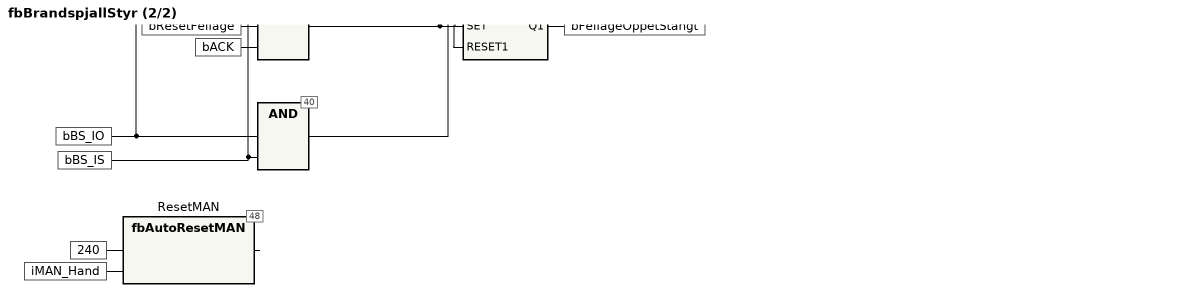
_CFC_ (* Continuous Function Chart, elements in execution order *)
(* **********************************************MOTIONERING********************************************** *)
(* **********************************************FELLÄGE SPJÄLL********************************************** *)
#0 OR(bManover, MotionManover)
#1 DELAY1:fbDelayedAlarmMinutes(_bLarm: bKomfel, _iMinutes: iKomfel_FL)
#2 AND(#0, NOT #1.bDelayedAlarm, NOT BrytManover)
#3 OVERRIDE:fbManualOverride(_bAuto: #2, _iMAN: iMAN_Hand, _iLM_Delay: iMAN_FL)
#4 bLM <= #3._bLM_DELAYED
#5 AND(#3._bStart, NOT bBRAND)
#6 bManoverUt <= #5
#7 PulsaMotionsKommando:TP(IN: bMotion, PT: t#1s)
#8 bResetFellage <= #7.Q
#9 AND(bManover, NOT bBRAND, #7.Q)
#10 DelayResetMotion:TON(IN: NOT bMotion, PT: t#15m)
#11 OR(bBRAND, #10.Q, bAvslutaMot)
#12 Motion_oppet:RS(SET: #9, RESET1: #11)
#13 StartaMotionOppetSpjall <= #12.Q1
#14 AND(NOT bManover, NOT bBRAND, #7.Q)
#15 OR(bBRAND, #10.Q, bAvslutaMot)
#16 Motion_stangt:RS(SET: #14, RESET1: #15)
#17 StartaMotionStangtSpjall <= #16.Q1
#18 OR(#12.Q1, #16.Q1)
#19 bMotionAktiv <= #18
#20 DelayMotOppet:TON(IN: StartaMotionOppetSpjall, PT: t#1s)
#21 Trig_bryt_man:R_TRIG(CLK: #20.Q)
#22 OR(bFellageStangerEJ, bBS_IS)
#23 DelayResetMotOppet:TON(IN: #22, PT: t#1s)
#24 Motion_oppet_bryt:SR(SET1: #21.Q, RESET: #23.Q)
#25 BrytManover <= #24.Q1
#26 AND(#24.Q1, #22)
#27 DelayMotStangt:TON(IN: StartaMotionStangtSpjall, PT: t#1s)
#28 Trig_man:R_TRIG(CLK: #27.Q)
#29 OR(bFellageOppnarEJ, bBS_IO)
#30 DelayResetMotStangt:TON(IN: #29, PT: t#1s)
#31 Motion_stangt_manover:SR(SET1: #28.Q, RESET: #30.Q)
#32 MotionManover <= #31.Q1
#33 AND(#31.Q1, #29)
#34 OR(#26, #33)
#35 bAvslutaMot <= #34
#36 AND(bManoverUt, NOT bBS_IO)
#37 DELAY2:fbDelayedAlarmSeconds(_bLarm: #36, _iSeconds: iBS_IO_FL)
#38 AND(NOT bManoverUt, NOT bBS_IS)
#39 DELAY3:fbDelayedAlarmSeconds(_bLarm: #38, _iSeconds: iBS_IS_FL)
#40 AND(bBS_IO, bBS_IS)
#41 OR(bResetFellage, bACK)
#42 SETRES1:RS(SET: #37.fDelayedAlarm2, RESET1: #41)
#43 bFellageOppnarEJ <= #42.Q1
#44 SETRES2:RS(SET: #39.fDelayedAlarm2, RESET1: #41)
#45 bFellageStangerEJ <= #44.Q1
#46 SETRES3:RS(SET: #40, RESET1: #41)
#47 bFellageOppetStangt <= #46.Q1
#48 ResetMAN:fbAutoResetMAN(240, iMAN_Hand)
_END_CFC_
END_FUNCTION_BLOCK

(* POU xEgna Funktionsblock/fbAutoResetMAN, CFC *)
FUNCTION_BLOCK fbAutoResetMAN
VAR_IN_OUT
	iMAN				:INT;

END_VAR
VAR_INPUT
	iResetDelay		:INT;

END_VAR
VAR_OUTPUT
END_VAR
VAR
	ResetDelay: TON;
END_VAR
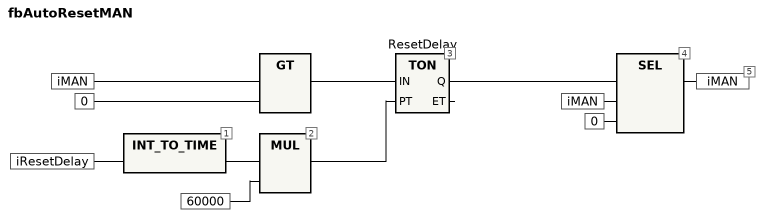
_CFC_ (* Continuous Function Chart, elements in execution order *)
#0 GT(iMAN, 0)
#1 INT_TO_TIME(iResetDelay)
#2 MUL(#1, 60000)
#3 ResetDelay:TON(IN: #0, PT: #2)
#4 SEL(#3.Q, iMAN, 0)
#5 iMAN <= #4
_END_CFC_
(* the same logic as Structured Text *)
ResetDelay(IN := iMAN > 0, PT := INT_TO_TIME(iResetDelay) * 60000);
iMAN := SEL(ResetDelay.Q, iMAN, 0);
END_FUNCTION_BLOCK

(* POU SYSTEM/Brandspjäll/HD71_BS201_BS202/HUS2_AS01_LB03_BS201_202, FAI *)
PROGRAM HUS2_AS01_LB03_BS201_202

VAR_INPUT
	bManover	 	:BOOL;
	bBRAND		:BOOL;
	bMotion		:BOOL;
	bKomfel		:BOOL;
END_VAR

VAR
	_bSetDefaultLocal: BOOL;

	SetAlarmDelay: FB_HVACPersistent_Int;
	SetAlarmDelay2: FB_HVACPersistent_Int;
	SetAlarmDelay3: FB_HVACPersistent_Int;
	SetAlarmDelay4: FB_HVACPersistent_Int;

	SpjallStyr: fbBrandspjallStyr2BS;

	ResetACK: fbBool_Reset;
	ResetACK2: fbBool_Reset;


END_VAR
(* body not read: cfc116 *)
END_PROGRAM

(* POU xEgna Funktionsblock/fbBrandspjallStyr2BS, CFC *)
FUNCTION_BLOCK fbBrandspjallStyr2BS
VAR_INPUT
	bManover						:BOOL;

	iMAN_FL1					:INT;
	bBS_IO1						:BOOL;
	iBS_IO_FL1					:INT;
	bBS_IS1						:BOOL;
	iBS_IS_FL1					:INT;
	bACK1						:BOOL;

	iMAN_FL2					:INT;
	bBS_IO2						:BOOL;
	iBS_IO_FL2					:INT;
	bBS_IS2						:BOOL;
	iBS_IS_FL2					:INT;
	bACK2						:BOOL;

	bBRAND						:BOOL;
	bKomfel						:BOOL;
	iKomfel_FL					:INT;
	bMotion						:BOOL;


END_VAR

VAR_IN_OUT
	iMAN_Hand1					:INT;
	iMAN_Hand2					:INT;
END_VAR

VAR_OUTPUT
	bManoverUt					:BOOL;
	bMotionAktiv					:BOOL;
	bLM1							:BOOL;
	bFellageOppnarEJ1			:BOOL;
	bFellageStangerEJ1			:BOOL;
	bFellageOppetStangt1			:BOOL;
	bLM2							:BOOL;
	bFellageOppnarEJ2			:BOOL;
	bFellageStangerEJ2			:BOOL;
	bFellageOppetStangt2			:BOOL;

END_VAR

VAR

	BrytManover: BOOL;
	MotionManover: BOOL;
	StartaMotionOppetSpjall: BOOL;
	StartaMotionStangtSpjall: BOOL;
	bResetFellage: BOOL;
	bAvslutaMot: BOOL;

	OVERRIDE1: fbManualOverride;
	ResetMAN1: fbAutoResetMAN;
	OVERRIDE2: fbManualOverride;
	ResetMAN2: fbAutoResetMAN;
	PulsaMotionsKommando: TP;
	DelayResetMotion: TON;

	DELAY1: fbDelayedAlarmMinutes;
	DELAY2: fbDelayedAlarmSeconds;
	DELAY3: fbDelayedAlarmSeconds;
	DELAY4: fbDelayedAlarmSeconds;
	DELAY5: fbDelayedAlarmSeconds;

	SETRES1: RS;
	SETRES2: RS;
	SETRES3: RS;
	SETRES4: RS;
	SETRES5: RS;
	SETRES6: RS;

	Motion_oppet: RS;
	Motion_oppet_bryt: SR;
	DelayMotOppet: TON;
	Trig_bryt_man: R_TRIG;
	DelayResetMotOppet: TON;

	Motion_stangt: RS;
	Motion_stangt_manover: SR;
	DelayMotStangt: TON;
	Trig_man: R_TRIG;
	DelayResetMotStangt: TON;


END_VAR
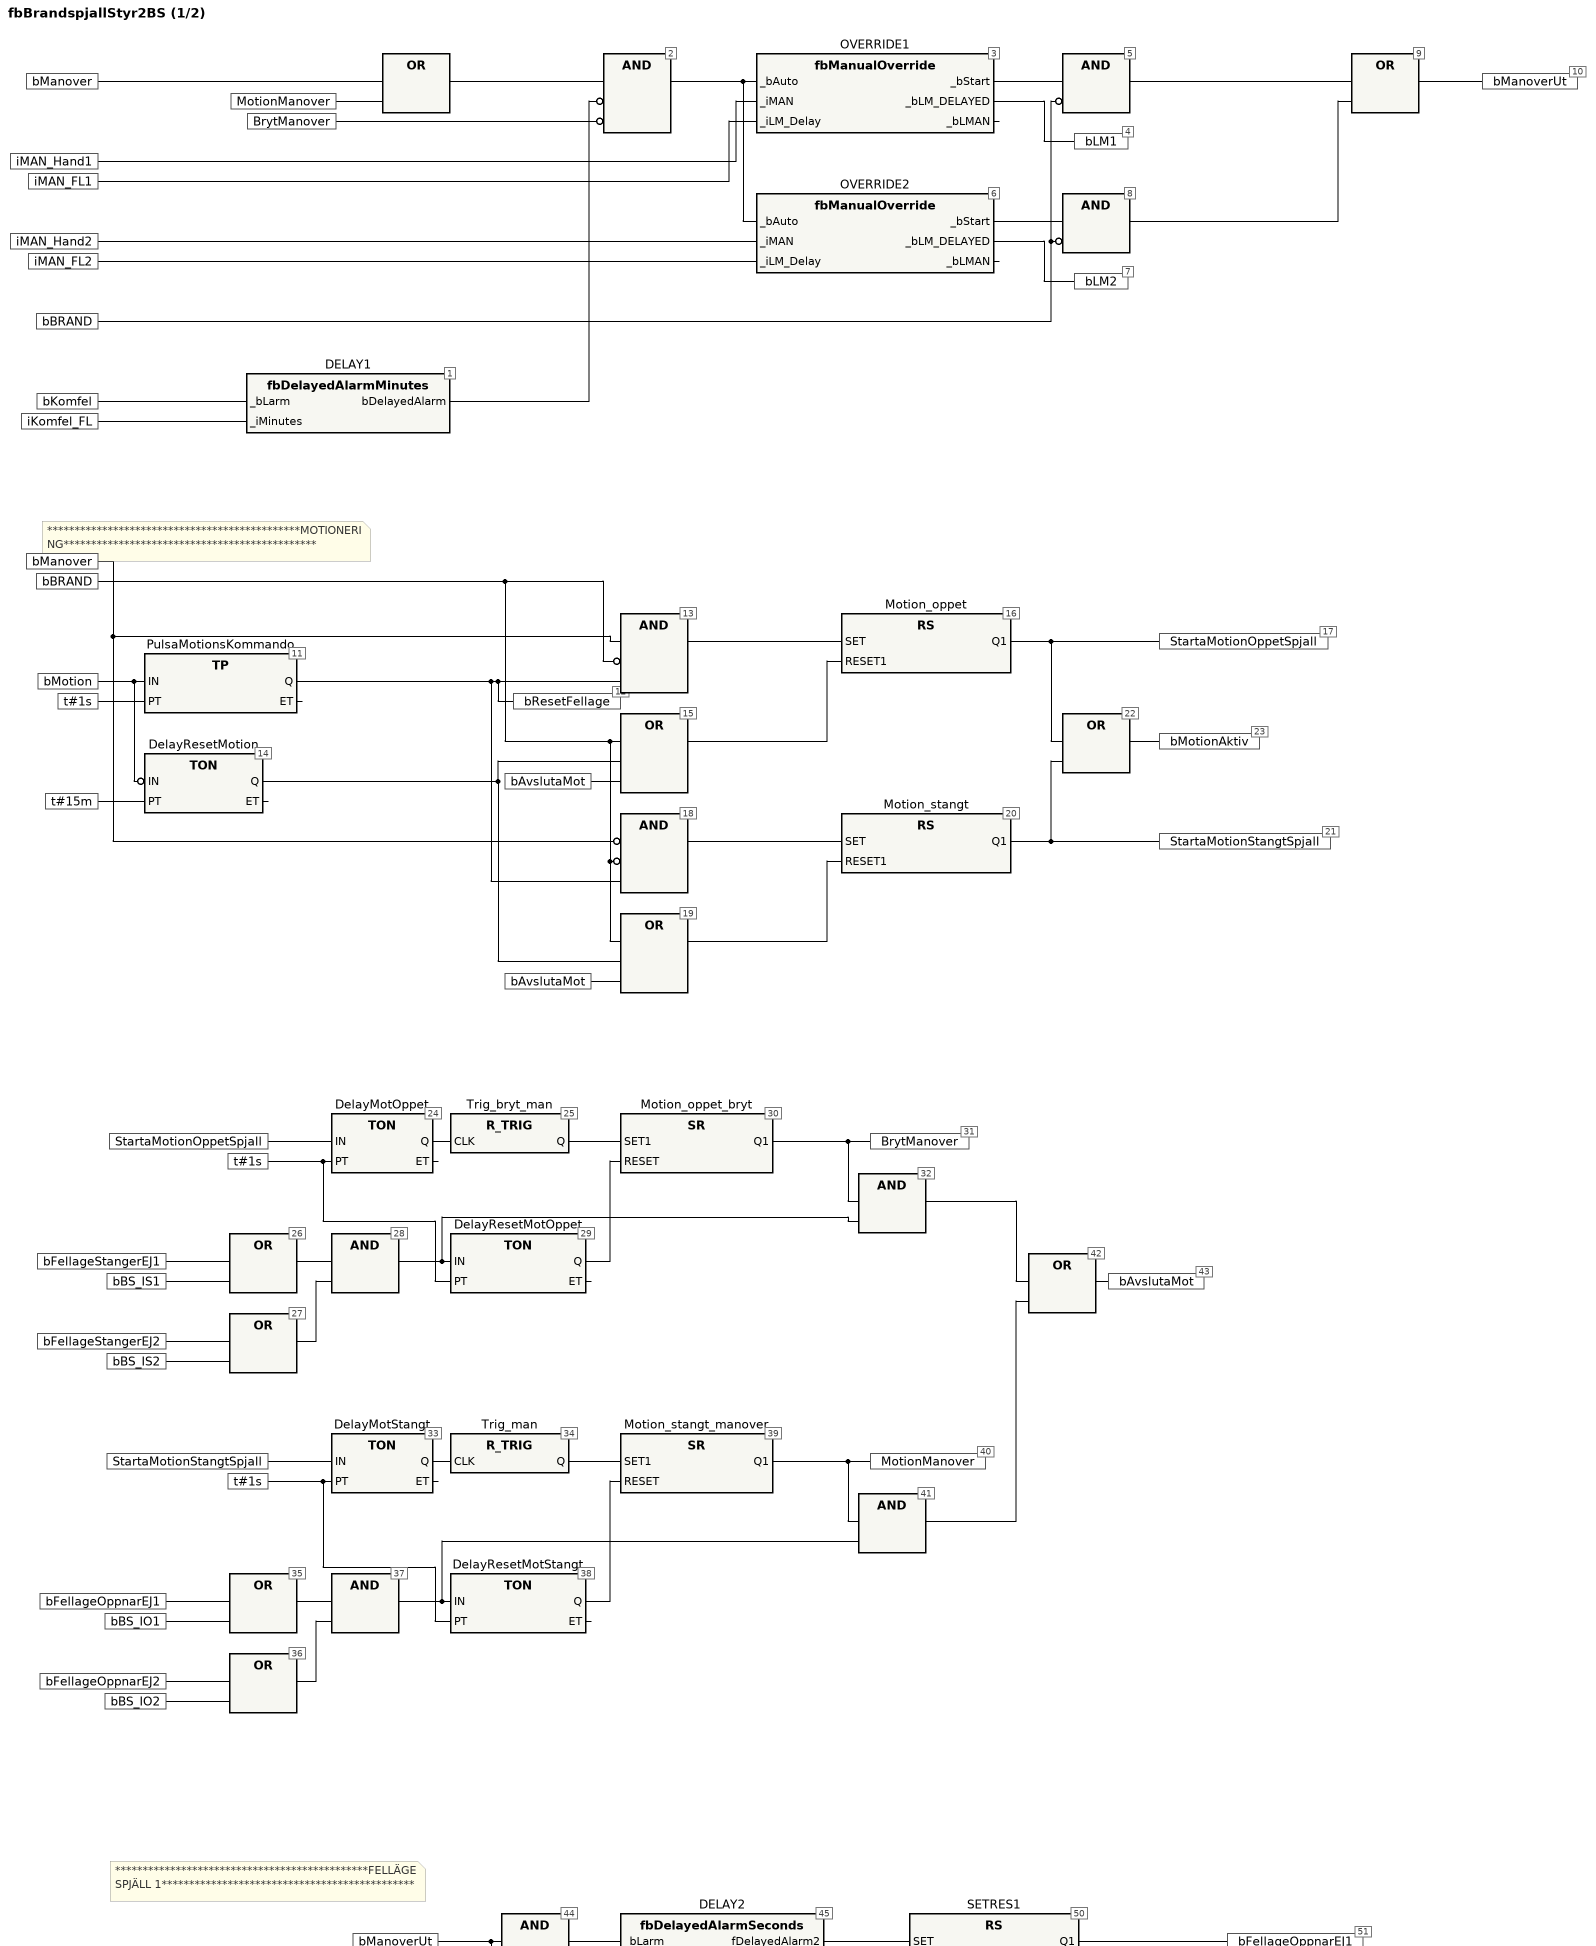
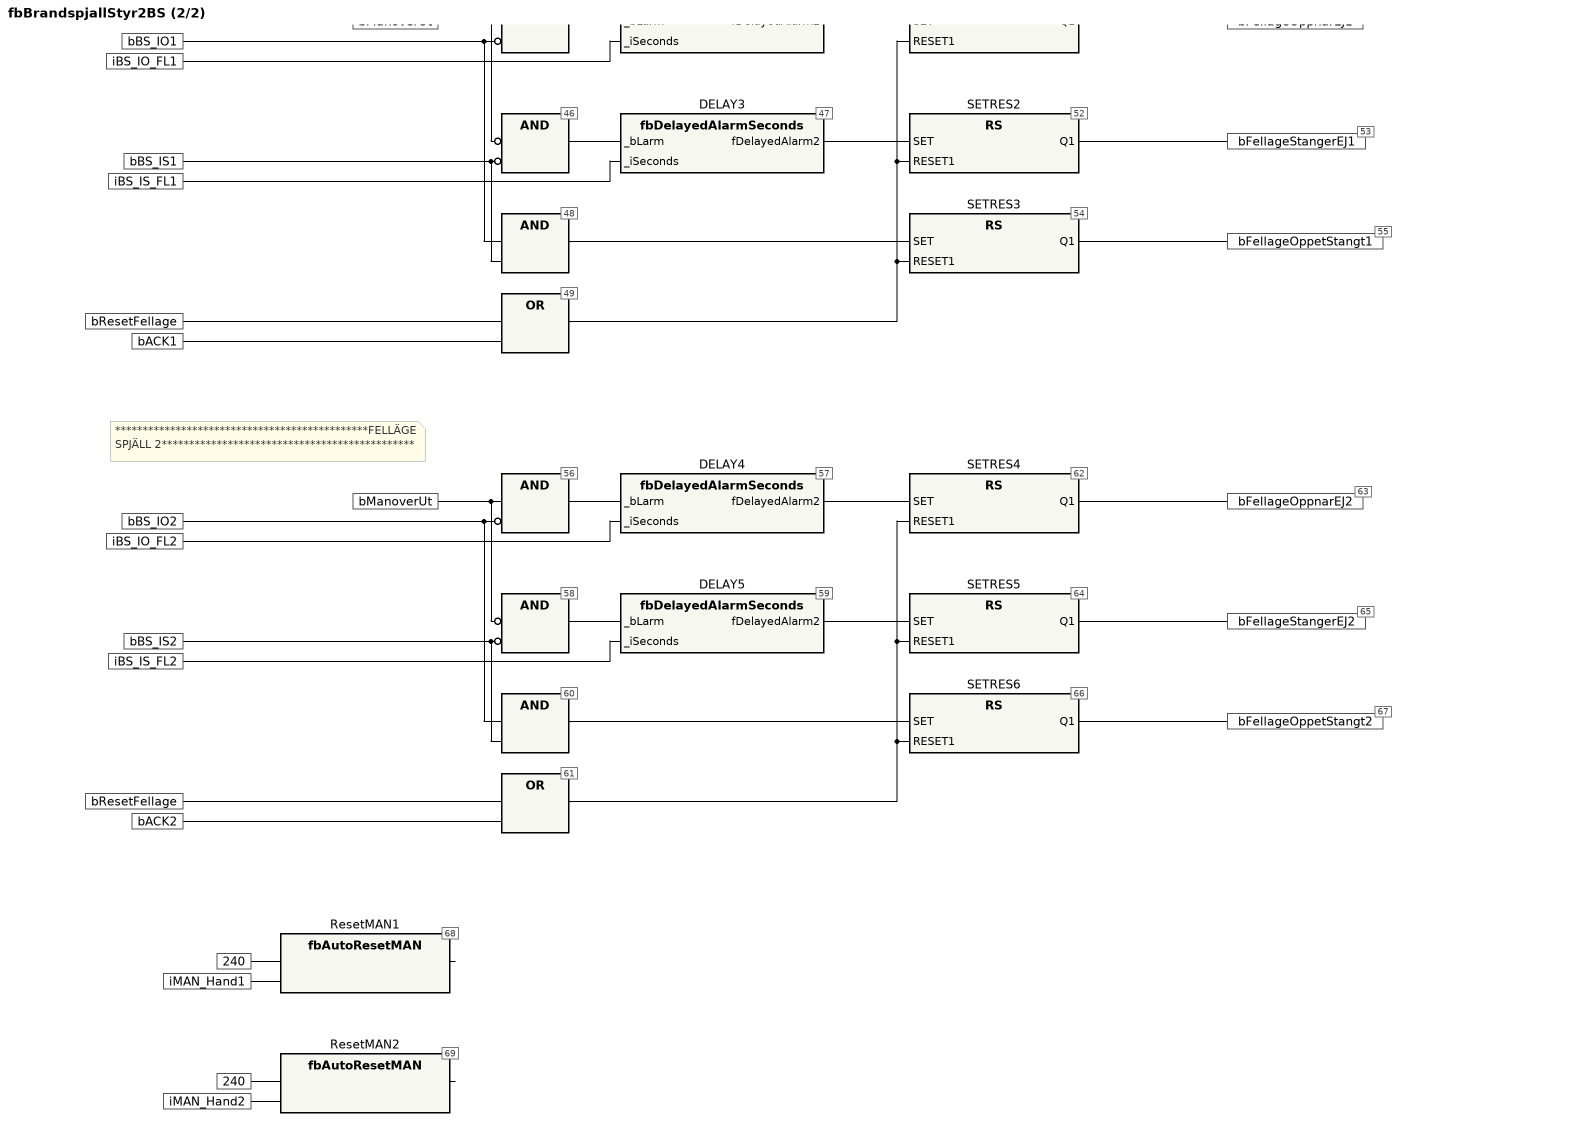
_CFC_ (* Continuous Function Chart, elements in execution order *)
(* **********************************************FELLÄGE SPJÄLL 2********************************************** *)
(* **********************************************FELLÄGE SPJÄLL 1********************************************** *)
(* **********************************************MOTIONERING********************************************** *)
#0 OR(bManover, MotionManover)
#1 DELAY1:fbDelayedAlarmMinutes(_bLarm: bKomfel, _iMinutes: iKomfel_FL)
#2 AND(#0, NOT #1.bDelayedAlarm, NOT BrytManover)
#3 OVERRIDE1:fbManualOverride(_bAuto: #2, _iMAN: iMAN_Hand1, _iLM_Delay: iMAN_FL1)
#4 bLM1 <= #3._bLM_DELAYED
#5 AND(#3._bStart, NOT bBRAND)
#6 OVERRIDE2:fbManualOverride(_bAuto: #2, _iMAN: iMAN_Hand2, _iLM_Delay: iMAN_FL2)
#7 bLM2 <= #6._bLM_DELAYED
#8 AND(#6._bStart, NOT bBRAND)
#9 OR(#5, #8)
#10 bManoverUt <= #9
#11 PulsaMotionsKommando:TP(IN: bMotion, PT: t#1s)
#12 bResetFellage <= #11.Q
#13 AND(bManover, NOT bBRAND, #11.Q)
#14 DelayResetMotion:TON(IN: NOT bMotion, PT: t#15m)
#15 OR(bBRAND, #14.Q, bAvslutaMot)
#16 Motion_oppet:RS(SET: #13, RESET1: #15)
#17 StartaMotionOppetSpjall <= #16.Q1
#18 AND(NOT bManover, NOT bBRAND, #11.Q)
#19 OR(bBRAND, #14.Q, bAvslutaMot)
#20 Motion_stangt:RS(SET: #18, RESET1: #19)
#21 StartaMotionStangtSpjall <= #20.Q1
#22 OR(#16.Q1, #20.Q1)
#23 bMotionAktiv <= #22
#24 DelayMotOppet:TON(IN: StartaMotionOppetSpjall, PT: t#1s)
#25 Trig_bryt_man:R_TRIG(CLK: #24.Q)
#26 OR(bFellageStangerEJ1, bBS_IS1)
#27 OR(bFellageStangerEJ2, bBS_IS2)
#28 AND(#26, #27)
#29 DelayResetMotOppet:TON(IN: #28, PT: t#1s)
#30 Motion_oppet_bryt:SR(SET1: #25.Q, RESET: #29.Q)
#31 BrytManover <= #30.Q1
#32 AND(#30.Q1, #28)
#33 DelayMotStangt:TON(IN: StartaMotionStangtSpjall, PT: t#1s)
#34 Trig_man:R_TRIG(CLK: #33.Q)
#35 OR(bFellageOppnarEJ1, bBS_IO1)
#36 OR(bFellageOppnarEJ2, bBS_IO2)
#37 AND(#35, #36)
#38 DelayResetMotStangt:TON(IN: #37, PT: t#1s)
#39 Motion_stangt_manover:SR(SET1: #34.Q, RESET: #38.Q)
#40 MotionManover <= #39.Q1
#41 AND(#39.Q1, #37)
#42 OR(#32, #41)
#43 bAvslutaMot <= #42
#44 AND(bManoverUt, NOT bBS_IO1)
#45 DELAY2:fbDelayedAlarmSeconds(_bLarm: #44, _iSeconds: iBS_IO_FL1)
#46 AND(NOT bManoverUt, NOT bBS_IS1)
#47 DELAY3:fbDelayedAlarmSeconds(_bLarm: #46, _iSeconds: iBS_IS_FL1)
#48 AND(bBS_IO1, bBS_IS1)
#49 OR(bResetFellage, bACK1)
#50 SETRES1:RS(SET: #45.fDelayedAlarm2, RESET1: #49)
#51 bFellageOppnarEJ1 <= #50.Q1
#52 SETRES2:RS(SET: #47.fDelayedAlarm2, RESET1: #49)
#53 bFellageStangerEJ1 <= #52.Q1
#54 SETRES3:RS(SET: #48, RESET1: #49)
#55 bFellageOppetStangt1 <= #54.Q1
#56 AND(bManoverUt, NOT bBS_IO2)
#57 DELAY4:fbDelayedAlarmSeconds(_bLarm: #56, _iSeconds: iBS_IO_FL2)
#58 AND(NOT bManoverUt, NOT bBS_IS2)
#59 DELAY5:fbDelayedAlarmSeconds(_bLarm: #58, _iSeconds: iBS_IS_FL2)
#60 AND(bBS_IO2, bBS_IS2)
#61 OR(bResetFellage, bACK2)
#62 SETRES4:RS(SET: #57.fDelayedAlarm2, RESET1: #61)
#63 bFellageOppnarEJ2 <= #62.Q1
#64 SETRES5:RS(SET: #59.fDelayedAlarm2, RESET1: #61)
#65 bFellageStangerEJ2 <= #64.Q1
#66 SETRES6:RS(SET: #60, RESET1: #61)
#67 bFellageOppetStangt2 <= #66.Q1
#68 ResetMAN1:fbAutoResetMAN(240, iMAN_Hand1)
#69 ResetMAN2:fbAutoResetMAN(240, iMAN_Hand2)
_END_CFC_
END_FUNCTION_BLOCK

(* POU SYSTEM/Brandspjäll/HD72_BS203/HUS2_AS01_LB03_BS203, FAI *)
PROGRAM HUS2_AS01_LB03_BS203

VAR_INPUT
	bManover	 	:BOOL;
	bBRAND		:BOOL;
	bMotion		:BOOL;
	bKomfel		:BOOL;
END_VAR

VAR
	_bSetDefaultLocal: BOOL;

	SetAlarmDelay: FB_HVACPersistent_Int;
	SetAlarmDelay2: FB_HVACPersistent_Int;

	SpjallStyr: fbBrandspjallStyr;

	ResetACK: fbBool_Reset;
END_VAR
(* body not read: cfc116 *)
END_PROGRAM

(* POU SYSTEM/Brandspjäll/HD74_BS205_BS206_BS207/HUS3_AL02_LB04_BS205_206_207, FAI *)
PROGRAM HUS3_AL02_LB04_BS205_206_207

VAR_INPUT
	bManover	 	:BOOL;
	bBRAND		:BOOL;
	bMotion		:BOOL;
	bKomfel		:BOOL;
END_VAR

VAR
	_bSetDefaultLocal: BOOL;

	SetAlarmDelay: FB_HVACPersistent_Int;
	SetAlarmDelay2: FB_HVACPersistent_Int;
	SetAlarmDelay3: FB_HVACPersistent_Int;
	SetAlarmDelay4: FB_HVACPersistent_Int;
	SetAlarmDelay5: FB_HVACPersistent_Int;
	SetAlarmDelay6: FB_HVACPersistent_Int;

	SpjallStyr: fbBrandspjallStyr3BS;

	ResetACK: fbBool_Reset;
	ResetACK2: fbBool_Reset;
	ResetACK3: fbBool_Reset;

END_VAR
(* body not read: cfc116 *)
END_PROGRAM

(* POU xEgna Funktionsblock/fbBrandspjallStyr3BS, CFC *)
FUNCTION_BLOCK fbBrandspjallStyr3BS
VAR_INPUT
	bManover						:BOOL;

	iMAN_FL1					:INT;
	bBS_IO1						:BOOL;
	iBS_IO_FL1					:INT;
	bBS_IS1						:BOOL;
	iBS_IS_FL1					:INT;
	bACK1						:BOOL;

	iMAN_FL2					:INT;
	bBS_IO2						:BOOL;
	iBS_IO_FL2					:INT;
	bBS_IS2						:BOOL;
	iBS_IS_FL2					:INT;
	bACK2						:BOOL;

	iMAN_FL3					:INT;
	bBS_IO3						:BOOL;
	iBS_IO_FL3					:INT;
	bBS_IS3						:BOOL;
	iBS_IS_FL3					:INT;
	bACK3						:BOOL;

	bBRAND						:BOOL;
	bKomfel						:BOOL;
	iKomfel_FL					:INT;
	bMotion						:BOOL;


END_VAR

VAR_IN_OUT
	iMAN_Hand1					:INT;
	iMAN_Hand2					:INT;
	iMAN_Hand3					:INT;

END_VAR

VAR_OUTPUT
	bManoverUt					:BOOL;
	bMotionAktiv					:BOOL;
	bLM1							:BOOL;
	bFellageOppnarEJ1			:BOOL;
	bFellageStangerEJ1			:BOOL;
	bFellageOppetStangt1			:BOOL;
	bLM2							:BOOL;
	bFellageOppnarEJ2			:BOOL;
	bFellageStangerEJ2			:BOOL;
	bFellageOppetStangt2			:BOOL;
	bLM3							:BOOL;
	bFellageOppnarEJ3			:BOOL;
	bFellageStangerEJ3			:BOOL;
	bFellageOppetStangt3			:BOOL;

END_VAR

VAR

	BrytManover: BOOL;
	MotionManover: BOOL;
	StartaMotionOppetSpjall: BOOL;
	StartaMotionStangtSpjall: BOOL;
	bResetFellage: BOOL;
	bAvslutaMot: BOOL;

	OVERRIDE1: fbManualOverride;
	ResetMAN1: fbAutoResetMAN;
	OVERRIDE2: fbManualOverride;
	ResetMAN2: fbAutoResetMAN;
	OVERRIDE3: fbManualOverride;
	ResetMAN3: fbAutoResetMAN;
	PulsaMotionsKommando: TP;
	DelayResetMotion: TON;

	DELAY1: fbDelayedAlarmMinutes;
	DELAY2: fbDelayedAlarmSeconds;
	DELAY3: fbDelayedAlarmSeconds;
	DELAY4: fbDelayedAlarmSeconds;
	DELAY5: fbDelayedAlarmSeconds;
	DELAY6: fbDelayedAlarmSeconds;
	DELAY7: fbDelayedAlarmSeconds;

	SETRES1: RS;
	SETRES2: RS;
	SETRES3: RS;
	SETRES4: RS;
	SETRES5: RS;
	SETRES6: RS;
	SETRES7: RS;
	SETRES8: RS;
	SETRES9: RS;

	Motion_oppet: RS;
	Motion_oppet_bryt: SR;
	DelayMotOppet: TON;
	Trig_bryt_man: R_TRIG;
	DelayResetMotOppet: TON;

	Motion_stangt: RS;
	Motion_stangt_manover: SR;
	DelayMotStangt: TON;
	Trig_man: R_TRIG;
	DelayResetMotStangt: TON;


END_VAR
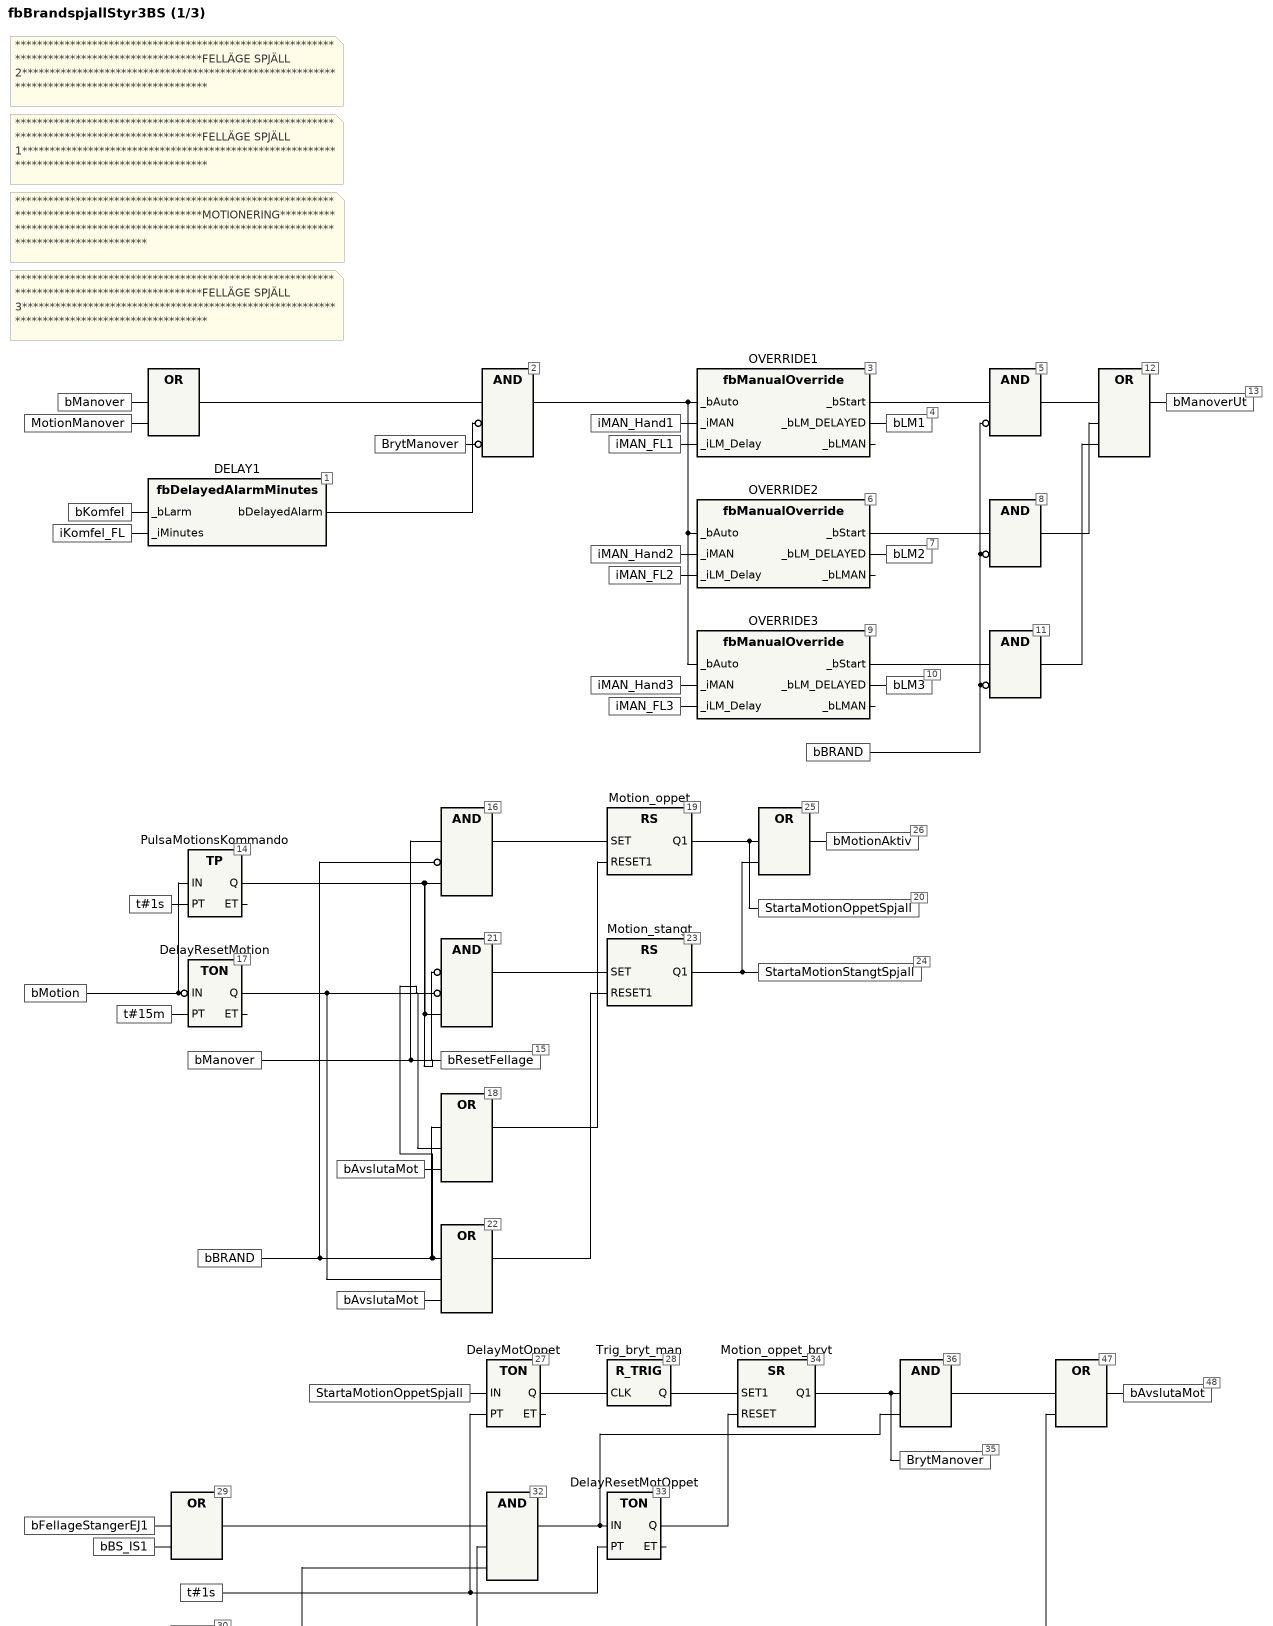
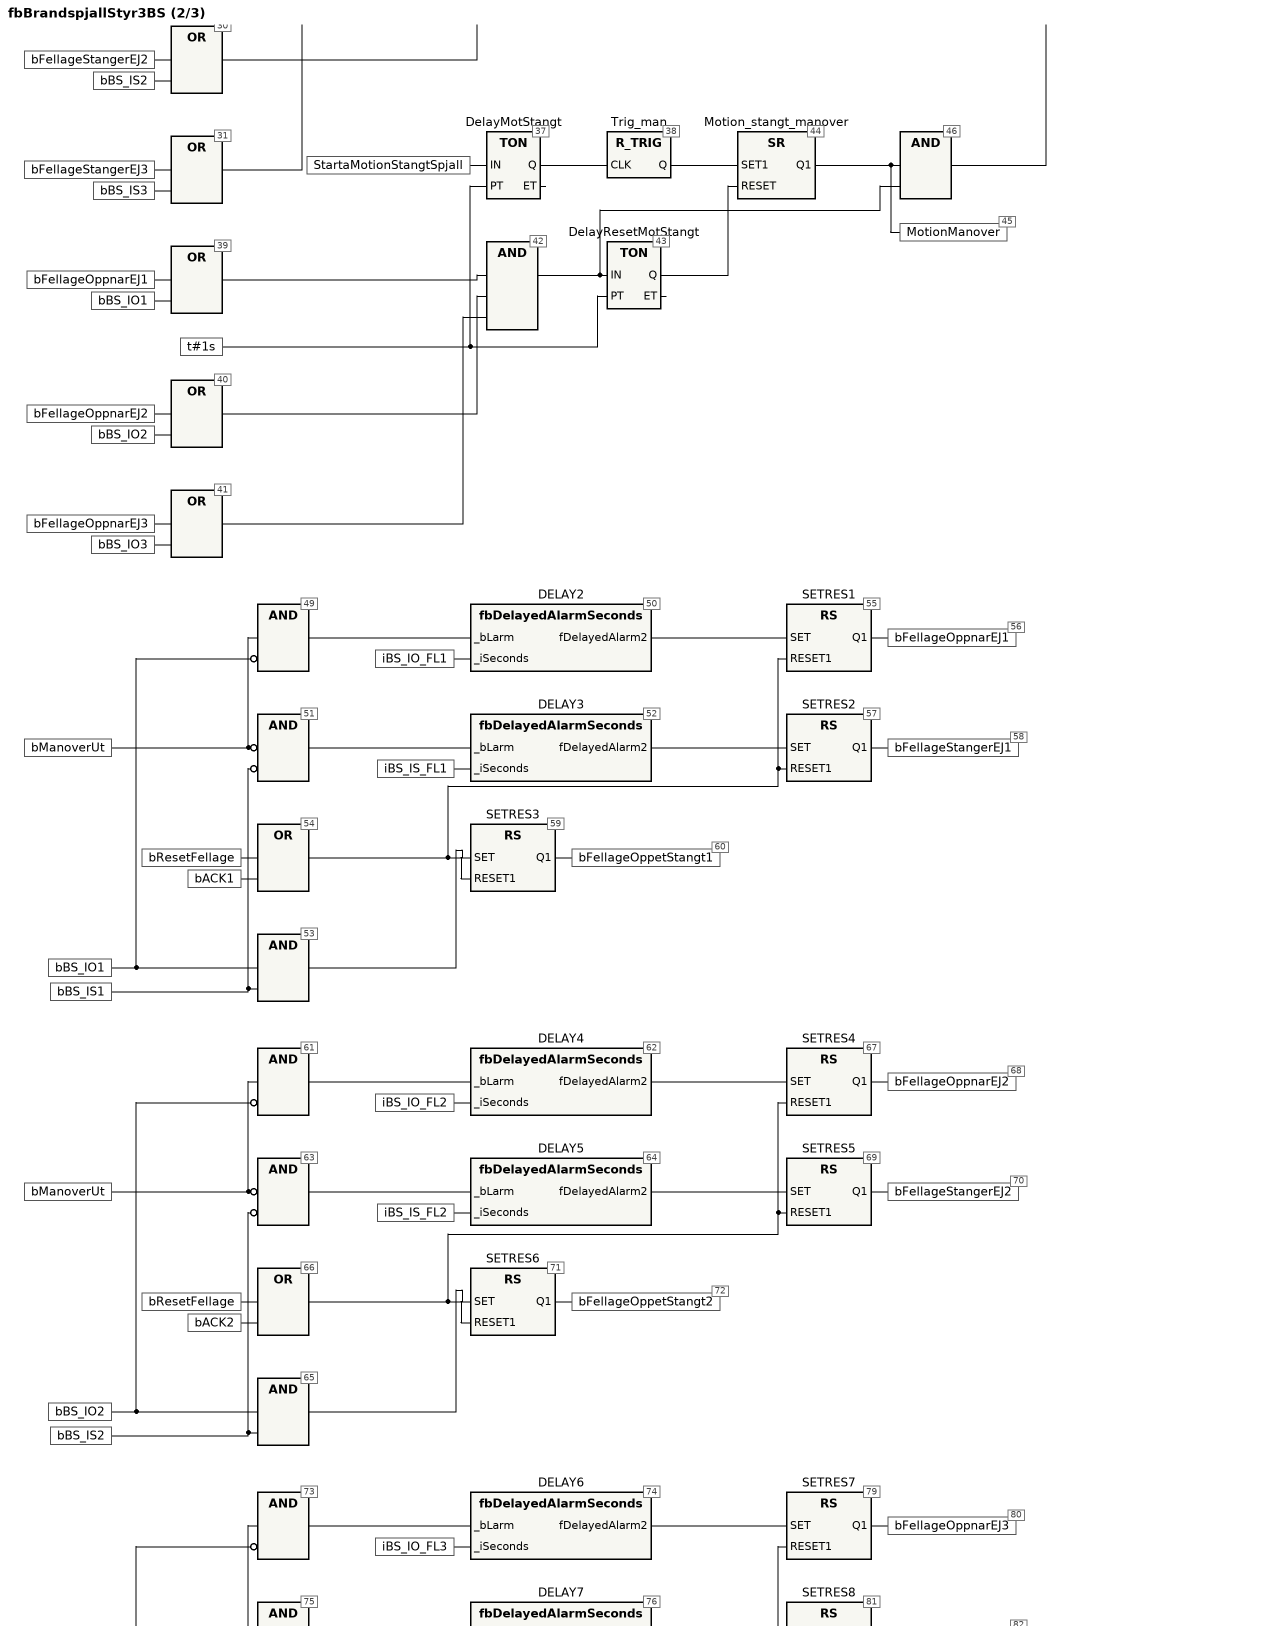
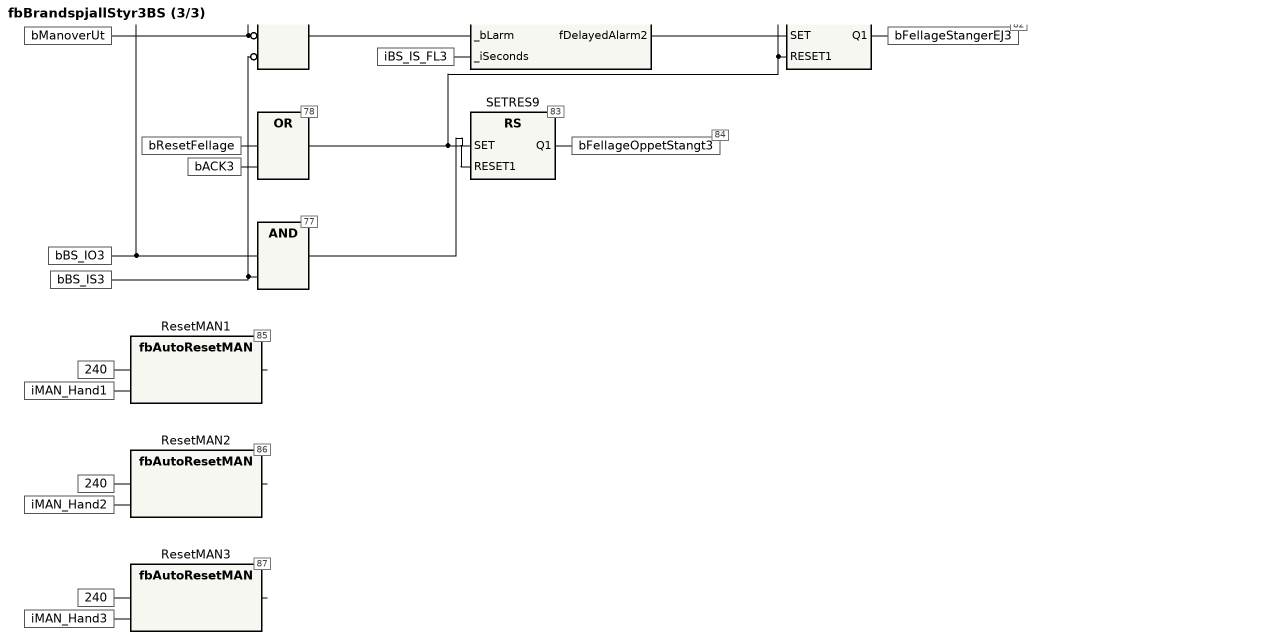
_CFC_ (* Continuous Function Chart, elements in execution order *)
(* ********************************************************************************************FELLÄGE SPJÄLL 2******************************************************************************************** *)
(* ********************************************************************************************FELLÄGE SPJÄLL 1******************************************************************************************** *)
(* ********************************************************************************************MOTIONERING******************************************************************************************** *)
(* ********************************************************************************************FELLÄGE SPJÄLL 3******************************************************************************************** *)
#0 OR(bManover, MotionManover)
#1 DELAY1:fbDelayedAlarmMinutes(_bLarm: bKomfel, _iMinutes: iKomfel_FL)
#2 AND(#0, NOT #1.bDelayedAlarm, NOT BrytManover)
#3 OVERRIDE1:fbManualOverride(_bAuto: #2, _iMAN: iMAN_Hand1, _iLM_Delay: iMAN_FL1)
#4 bLM1 <= #3._bLM_DELAYED
#5 AND(#3._bStart, NOT bBRAND)
#6 OVERRIDE2:fbManualOverride(_bAuto: #2, _iMAN: iMAN_Hand2, _iLM_Delay: iMAN_FL2)
#7 bLM2 <= #6._bLM_DELAYED
#8 AND(#6._bStart, NOT bBRAND)
#9 OVERRIDE3:fbManualOverride(_bAuto: #2, _iMAN: iMAN_Hand3, _iLM_Delay: iMAN_FL3)
#10 bLM3 <= #9._bLM_DELAYED
#11 AND(#9._bStart, NOT bBRAND)
#12 OR(#5, #8, #11)
#13 bManoverUt <= #12
#14 PulsaMotionsKommando:TP(IN: bMotion, PT: t#1s)
#15 bResetFellage <= #14.Q
#16 AND(bManover, NOT bBRAND, #14.Q)
#17 DelayResetMotion:TON(IN: NOT bMotion, PT: t#15m)
#18 OR(bBRAND, #17.Q, bAvslutaMot)
#19 Motion_oppet:RS(SET: #16, RESET1: #18)
#20 StartaMotionOppetSpjall <= #19.Q1
#21 AND(NOT bManover, NOT bBRAND, #14.Q)
#22 OR(bBRAND, #17.Q, bAvslutaMot)
#23 Motion_stangt:RS(SET: #21, RESET1: #22)
#24 StartaMotionStangtSpjall <= #23.Q1
#25 OR(#19.Q1, #23.Q1)
#26 bMotionAktiv <= #25
#27 DelayMotOppet:TON(IN: StartaMotionOppetSpjall, PT: t#1s)
#28 Trig_bryt_man:R_TRIG(CLK: #27.Q)
#29 OR(bFellageStangerEJ1, bBS_IS1)
#30 OR(bFellageStangerEJ2, bBS_IS2)
#31 OR(bFellageStangerEJ3, bBS_IS3)
#32 AND(#29, #30, #31)
#33 DelayResetMotOppet:TON(IN: #32, PT: t#1s)
#34 Motion_oppet_bryt:SR(SET1: #28.Q, RESET: #33.Q)
#35 BrytManover <= #34.Q1
#36 AND(#34.Q1, #32)
#37 DelayMotStangt:TON(IN: StartaMotionStangtSpjall, PT: t#1s)
#38 Trig_man:R_TRIG(CLK: #37.Q)
#39 OR(bFellageOppnarEJ1, bBS_IO1)
#40 OR(bFellageOppnarEJ2, bBS_IO2)
#41 OR(bFellageOppnarEJ3, bBS_IO3)
#42 AND(#39, #40, #41)
#43 DelayResetMotStangt:TON(IN: #42, PT: t#1s)
#44 Motion_stangt_manover:SR(SET1: #38.Q, RESET: #43.Q)
#45 MotionManover <= #44.Q1
#46 AND(#44.Q1, #42)
#47 OR(#36, #46)
#48 bAvslutaMot <= #47
#49 AND(bManoverUt, NOT bBS_IO1)
#50 DELAY2:fbDelayedAlarmSeconds(_bLarm: #49, _iSeconds: iBS_IO_FL1)
#51 AND(NOT bManoverUt, NOT bBS_IS1)
#52 DELAY3:fbDelayedAlarmSeconds(_bLarm: #51, _iSeconds: iBS_IS_FL1)
#53 AND(bBS_IO1, bBS_IS1)
#54 OR(bResetFellage, bACK1)
#55 SETRES1:RS(SET: #50.fDelayedAlarm2, RESET1: #54)
#56 bFellageOppnarEJ1 <= #55.Q1
#57 SETRES2:RS(SET: #52.fDelayedAlarm2, RESET1: #54)
#58 bFellageStangerEJ1 <= #57.Q1
#59 SETRES3:RS(SET: #53, RESET1: #54)
#60 bFellageOppetStangt1 <= #59.Q1
#61 AND(bManoverUt, NOT bBS_IO2)
#62 DELAY4:fbDelayedAlarmSeconds(_bLarm: #61, _iSeconds: iBS_IO_FL2)
#63 AND(NOT bManoverUt, NOT bBS_IS2)
#64 DELAY5:fbDelayedAlarmSeconds(_bLarm: #63, _iSeconds: iBS_IS_FL2)
#65 AND(bBS_IO2, bBS_IS2)
#66 OR(bResetFellage, bACK2)
#67 SETRES4:RS(SET: #62.fDelayedAlarm2, RESET1: #66)
#68 bFellageOppnarEJ2 <= #67.Q1
#69 SETRES5:RS(SET: #64.fDelayedAlarm2, RESET1: #66)
#70 bFellageStangerEJ2 <= #69.Q1
#71 SETRES6:RS(SET: #65, RESET1: #66)
#72 bFellageOppetStangt2 <= #71.Q1
#73 AND(bManoverUt, NOT bBS_IO3)
#74 DELAY6:fbDelayedAlarmSeconds(_bLarm: #73, _iSeconds: iBS_IO_FL3)
#75 AND(NOT bManoverUt, NOT bBS_IS3)
#76 DELAY7:fbDelayedAlarmSeconds(_bLarm: #75, _iSeconds: iBS_IS_FL3)
#77 AND(bBS_IO3, bBS_IS3)
#78 OR(bResetFellage, bACK3)
#79 SETRES7:RS(SET: #74.fDelayedAlarm2, RESET1: #78)
#80 bFellageOppnarEJ3 <= #79.Q1
#81 SETRES8:RS(SET: #76.fDelayedAlarm2, RESET1: #78)
#82 bFellageStangerEJ3 <= #81.Q1
#83 SETRES9:RS(SET: #77, RESET1: #78)
#84 bFellageOppetStangt3 <= #83.Q1
#85 ResetMAN1:fbAutoResetMAN(240, iMAN_Hand1)
#86 ResetMAN2:fbAutoResetMAN(240, iMAN_Hand2)
#87 ResetMAN3:fbAutoResetMAN(240, iMAN_Hand3)
_END_CFC_
END_FUNCTION_BLOCK

(* POU SYSTEM/Brandspjäll/HD75_BS208_BS209_BS210/HUS3_AL03_LB05_BS208_209_210, FAI *)
PROGRAM HUS3_AL03_LB05_BS208_209_210

VAR_INPUT
	bManover	 	:BOOL;
	bBRAND		:BOOL;
	bMotion		:BOOL;
	bKomfel		:BOOL;
END_VAR

VAR
	_bSetDefaultLocal: BOOL;

	SetAlarmDelay: FB_HVACPersistent_Int;
	SetAlarmDelay2: FB_HVACPersistent_Int;
	SetAlarmDelay3: FB_HVACPersistent_Int;
	SetAlarmDelay4: FB_HVACPersistent_Int;
	SetAlarmDelay5: FB_HVACPersistent_Int;
	SetAlarmDelay6: FB_HVACPersistent_Int;

	SpjallStyr: fbBrandspjallStyr3BS;

	ResetACK: fbBool_Reset;
	ResetACK2: fbBool_Reset;
	ResetACK3: fbBool_Reset;


END_VAR
(* body not read: cfc116 *)
END_PROGRAM

(* POU SYSTEM/VP1/HUS2_VP1, CFC *)
PROGRAM HUS2_VP1
VAR
	_bSetDefault_Plant:BOOL;
	_bReset_Plant:BOOL;

	SETRESET: SR;
	ACK_RESET: fbBool_Reset;
	SETRESET1: SR;
	SV_MQ41: REAL;
END_VAR
VAR (* helpers for the ST form of the networks *)
	_t25 : BOOL;
END_VAR
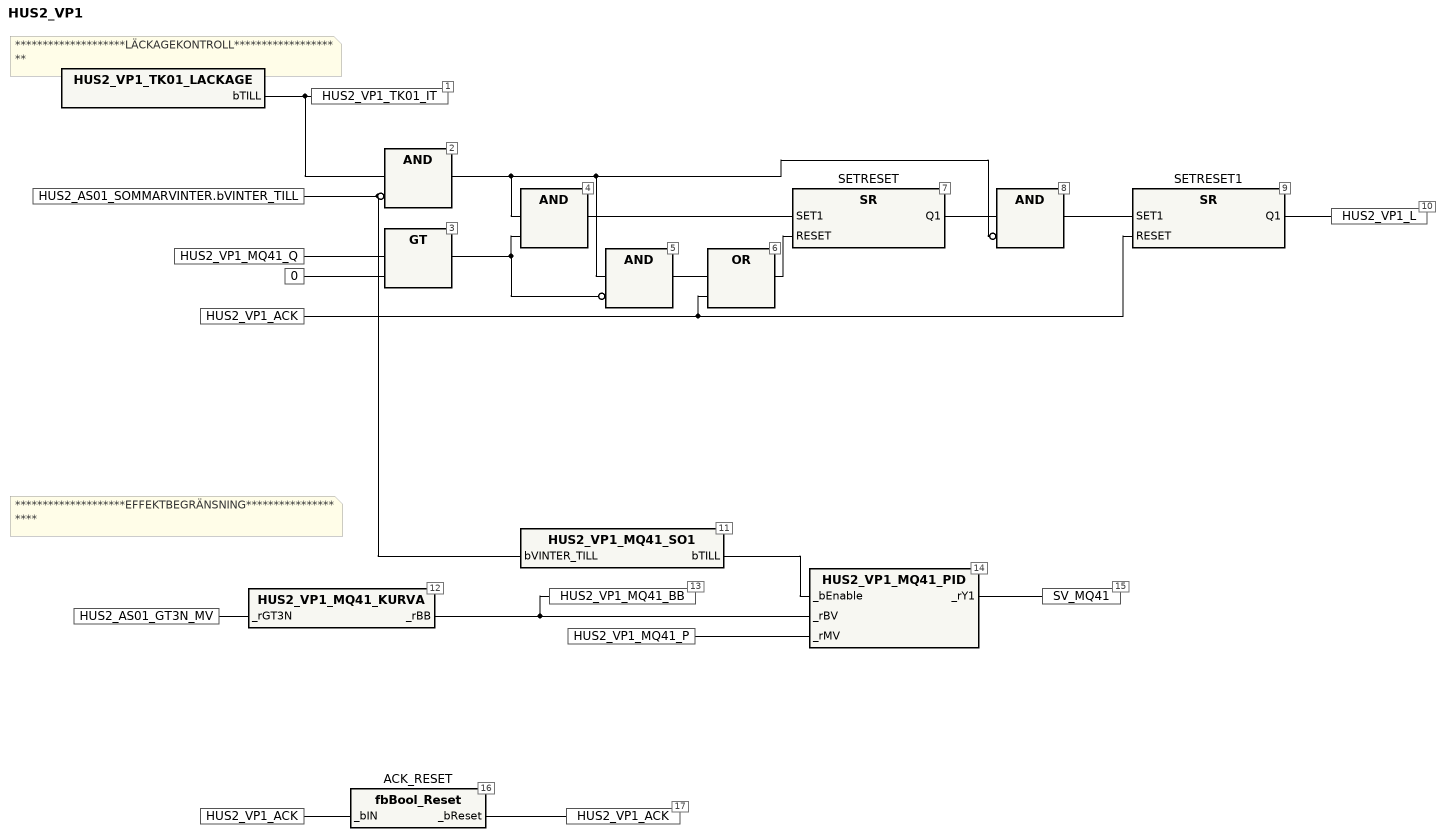
_CFC_ (* Continuous Function Chart, elements in execution order *)
(* ********************EFFEKTBEGRÄNSNING******************** *)
(* ********************LÄCKAGEKONTROLL******************** *)
#0 HUS2_VP1_TK01_LACKAGE()
#1 HUS2_VP1_TK01_IT <= #0.bTILL
#2 AND(#0.bTILL, NOT HUS2_AS01_SOMMARVINTER.bVINTER_TILL)
#3 GT(HUS2_VP1_MQ41_Q, 0)
#4 AND(#2, #3)
#5 AND(#2, NOT #3)
#6 OR(#5, HUS2_VP1_ACK)
#7 SETRESET:SR(SET1: #4, RESET: #6)
#8 AND(#7.Q1, NOT #2)
#9 SETRESET1:SR(SET1: #8, RESET: HUS2_VP1_ACK)
#10 HUS2_VP1_L <= #9.Q1
#11 HUS2_VP1_MQ41_SO1(bVINTER_TILL: HUS2_AS01_SOMMARVINTER.bVINTER_TILL)
#12 HUS2_VP1_MQ41_KURVA(_rGT3N: HUS2_AS01_GT3N_MV)
#13 HUS2_VP1_MQ41_BB <= #12._rBB
#14 HUS2_VP1_MQ41_PID(_bEnable: #11.bTILL, _rBV: #12._rBB, _rMV: HUS2_VP1_MQ41_P)
#15 SV_MQ41 <= #14._rY1
#16 ACK_RESET:fbBool_Reset(_bIN: HUS2_VP1_ACK)
#17 HUS2_VP1_ACK <= #16._bReset
_END_CFC_
(* the same logic as Structured Text *)
(* ********************EFFEKTBEGRÄNSNING******************** *)
(* ********************LÄCKAGEKONTROLL******************** *)
HUS2_VP1_TK01_LACKAGE();
HUS2_VP1_TK01_IT := HUS2_VP1_TK01_LACKAGE.bTILL;
_t25 := HUS2_VP1_TK01_LACKAGE.bTILL AND NOT HUS2_AS01_SOMMARVINTER.bVINTER_TILL;
SETRESET(SET1 := _t25 AND (HUS2_VP1_MQ41_Q > 0), RESET := (_t25 AND NOT (HUS2_VP1_MQ41_Q > 0)) OR HUS2_VP1_ACK);
SETRESET1(SET1 := SETRESET.Q1 AND NOT _t25, RESET := HUS2_VP1_ACK);
HUS2_VP1_L := SETRESET1.Q1;
HUS2_VP1_MQ41_SO1(bVINTER_TILL := HUS2_AS01_SOMMARVINTER.bVINTER_TILL);
HUS2_VP1_MQ41_KURVA(_rGT3N := HUS2_AS01_GT3N_MV);
HUS2_VP1_MQ41_BB := HUS2_VP1_MQ41_KURVA._rBB;
HUS2_VP1_MQ41_PID(_bEnable := HUS2_VP1_MQ41_SO1.bTILL, _rBV := HUS2_VP1_MQ41_KURVA._rBB, _rMV := HUS2_VP1_MQ41_P);
SV_MQ41 := HUS2_VP1_MQ41_PID._rY1;
ACK_RESET(_bIN := HUS2_VP1_ACK);
HUS2_VP1_ACK := ACK_RESET._bReset;
END_PROGRAM

(* POU SYSTEM/VP1/HUS2_VP1_TK01_LACKAGE, CFC *)
PROGRAM HUS2_VP1_TK01_LACKAGE

VAR
	AUTO_MAN: fbManualOverride;

END_VAR

VAR_OUTPUT
	bTILL			:BOOL;
END_VAR
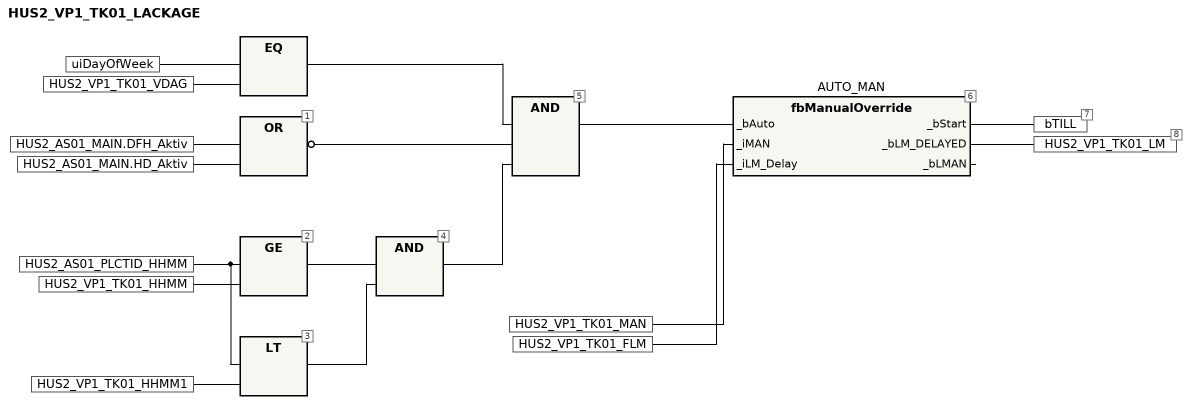
_CFC_ (* Continuous Function Chart, elements in execution order *)
#0 EQ(uiDayOfWeek, HUS2_VP1_TK01_VDAG)
#1 OR(HUS2_AS01_MAIN.DFH_Aktiv, HUS2_AS01_MAIN.HD_Aktiv)
#2 GE(HUS2_AS01_PLCTID_HHMM, HUS2_VP1_TK01_HHMM)
#3 LT(HUS2_AS01_PLCTID_HHMM, HUS2_VP1_TK01_HHMM1)
#4 AND(#2, #3)
#5 AND(#0, NOT #1, #4)
#6 AUTO_MAN:fbManualOverride(_bAuto: #5, _iMAN: HUS2_VP1_TK01_MAN, _iLM_Delay: HUS2_VP1_TK01_FLM)
#7 bTILL <= #6._bStart
#8 HUS2_VP1_TK01_LM <= #6._bLM_DELAYED
_END_CFC_
(* the same logic as Structured Text *)
AUTO_MAN(_bAuto := (uiDayOfWeek = HUS2_VP1_TK01_VDAG) AND NOT (HUS2_AS01_MAIN.DFH_Aktiv OR HUS2_AS01_MAIN.HD_Aktiv) AND ((HUS2_AS01_PLCTID_HHMM >= HUS2_VP1_TK01_HHMM) AND (HUS2_AS01_PLCTID_HHMM < HUS2_VP1_TK01_HHMM1)), _iMAN := HUS2_VP1_TK01_MAN, _iLM_Delay := HUS2_VP1_TK01_FLM);
bTILL := AUTO_MAN._bStart;
HUS2_VP1_TK01_LM := AUTO_MAN._bLM_DELAYED;
END_PROGRAM

(* POU SYSTEM/VP1/Begränsning/HUS2_VP1_MQ41_SO1, CFC *)
PROGRAM HUS2_VP1_MQ41_SO1
VAR
END_VAR


VAR_INPUT
	bVINTER_TILL		:BOOL;

END_VAR

VAR_OUTPUT
	bTILL: BOOL;

END_VAR
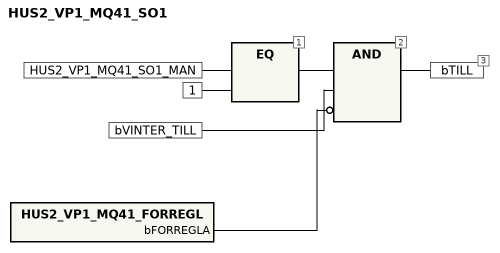
_CFC_ (* Continuous Function Chart, elements in execution order *)
#0 HUS2_VP1_MQ41_FORREGL()
#1 EQ(HUS2_VP1_MQ41_SO1_MAN, 1)
#2 AND(#1, bVINTER_TILL, NOT #0.bFORREGLA)
#3 bTILL <= #2
_END_CFC_
(* the same logic as Structured Text *)
HUS2_VP1_MQ41_FORREGL();
bTILL := (HUS2_VP1_MQ41_SO1_MAN = 1) AND bVINTER_TILL AND NOT HUS2_VP1_MQ41_FORREGL.bFORREGLA;
END_PROGRAM

(* POU SYSTEM/VP1/Begränsning/HUS2_VP1_MQ41_FORREGL, CFC *)
PROGRAM HUS2_VP1_MQ41_FORREGL
VAR
END_VAR
VAR_OUTPUT
	bFORREGLA: BOOL;
END_VAR
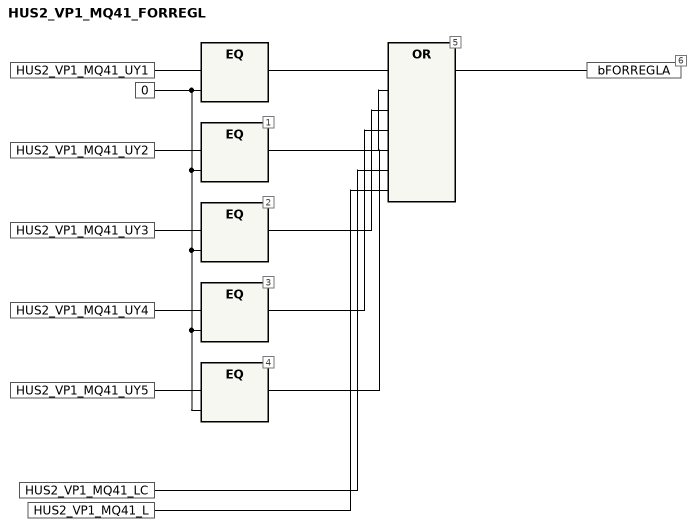
_CFC_ (* Continuous Function Chart, elements in execution order *)
#0 EQ(HUS2_VP1_MQ41_UY1, 0)
#1 EQ(HUS2_VP1_MQ41_UY2, 0)
#2 EQ(HUS2_VP1_MQ41_UY3, 0)
#3 EQ(HUS2_VP1_MQ41_UY4, 0)
#4 EQ(HUS2_VP1_MQ41_UY5, 0)
#5 OR(#0, #1, #2, #3, #4, HUS2_VP1_MQ41_LC, HUS2_VP1_MQ41_L)
#6 bFORREGLA <= #5
_END_CFC_
(* the same logic as Structured Text *)
bFORREGLA := (HUS2_VP1_MQ41_UY1 = 0) OR (HUS2_VP1_MQ41_UY2 = 0) OR (HUS2_VP1_MQ41_UY3 = 0) OR (HUS2_VP1_MQ41_UY4 = 0) OR (HUS2_VP1_MQ41_UY5 = 0) OR HUS2_VP1_MQ41_LC OR HUS2_VP1_MQ41_L;
END_PROGRAM

(* POU SYSTEM/VP1/Begränsning/HUS2_VP1_MQ41_KURVA, FAI *)
PROGRAM HUS2_VP1_MQ41_KURVA
VAR
(****************************************** heating curve **********************************************************************************************************************)

	_bSetDefaultHC			:BOOL;


	fbScale_n:			FB_HVACScale_nPoint;
	_bErrParam:			BOOL;								(*ParameterError*)
	stScaleParameter:	ST_HVACParameterScale_nPoint	;	(*Parameter struktur på antal brutpunkter*)


	fbTemp1:	FB_HVACPersistent_Real;
	fbTemp2:	FB_HVACPersistent_Real;
	fbTemp3:	FB_HVACPersistent_Real;
	fbTemp4:	FB_HVACPersistent_Real;
	fbTemp5:	FB_HVACPersistent_Real;

	fbOutsideTemp1:	FB_HVACPersistent_Real;
	fbOutsideTemp2:	FB_HVACPersistent_Real;
	fbOutsideTemp3:	FB_HVACPersistent_Real;
	fbOutsideTemp4:	FB_HVACPersistent_Real;
	fbOutsideTemp5:	FB_HVACPersistent_Real;
	BB_min: FB_HVACPersistent_Real;
	BB_max: FB_HVACPersistent_Real;

END_VAR

VAR_INPUT
	_rGT3N	:REAL; (*Utegivare*)

END_VAR

VAR_OUTPUT
	_rBB		:LREAL;
END_VAR
(* body not read: cfc97 *)
END_PROGRAM

(* POU SYSTEM/VP1/Begränsning/HUS2_VP1_MQ41_PID, FAI *)
PROGRAM HUS2_VP1_MQ41_PID

VAR_INPUT
	_bEnable		:BOOL;
	_rBV			:REAL;
	_rMV			:REAL;
END_VAR

VAR_OUTPUT
	_rY1                         : REAL;
END_VAR


VAR
	_bSetDefaultPID:BOOL;
	_bReset_Local:BOOL;


	SVX: FB_HVACPIDCtrl;
	eDataSecurityType         : E_HVACDataSecurityType;
	rInitialValue            : REAL;
	bResetController          : BOOL;
	_eCtrlMode				:E_HVACCtrlMode;(*
									eHVACCtrlMode_Auto      := 0,
								   	eHVACCtrlMode_Manual   := 1 *)
	_rOverrideValue			:REAL;(* controller output rY in operating mode eCtrlMode =1 *)
	rXW                        : REAL;
	bMaxLimit                  : BOOL;
	bMinLimit                  : BOOL;
	bActive                    : BOOL;
	bARWactive                 : BOOL;
	eState                     : E_HVACState;
	bError                     : BOOL;
	eErrorCode                 : E_HVACErrorCodes;
	bInvalidParameter          : BOOL;

	bDirection              : BOOL;
	_rKP: REAL;
	_rCH: REAL;
	tTi                     : TIME;
	tTv                     : TIME;
	tTd                     : TIME;

	rYMin                   : REAL;
	rYMax                   : REAL;

	CI: fbBer_PID_inst;
	CS: fbBer_PID_inst;
	CD: fbBer_PID_inst;

	fbPersistent_CH: FB_HVACPersistent_Real;
	fbPersistent_CP: FB_HVACPersistent_Real;
	fbPersistent_CI: FB_HVACPersistent_Real;
	fbPersistent_CS: FB_HVACPersistent_Real;
	fbPersistent_CD: FB_HVACPersistent_Real;
	LM_DELAY: fbDelayedAlarmMinutes;


	SLIDE: FB_HVACTimeAverage;
	udiNumOfElem   : UDINT:=40;
END_VAR
(* body not read: cfc97 *)
END_PROGRAM

(* POU xEgna Funktionsblock/fbBer_PID_inst, CFC *)
FUNCTION_BLOCK fbBer_PID_inst
VAR_INPUT
	_rIN:REAL;
END_VAR
VAR_OUTPUT
	_tOUT:TIME;
END_VAR
VAR
END_VAR
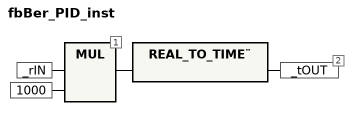
_CFC_ (* Continuous Function Chart, elements in execution order *)
#0 REAL_TO_TIME¨(#1)
#1 MUL(_rIN, 1000)
#2 _tOUT <= #0
_END_CFC_
END_FUNCTION_BLOCK

(* POU SYSTEM/VS1/HUS2_VS1, CFC *)
PROGRAM HUS2_VS1
VAR
	_bSetDefault_Plant		:BOOL;
	_bReset_Plant				:BOOL;

END_VAR
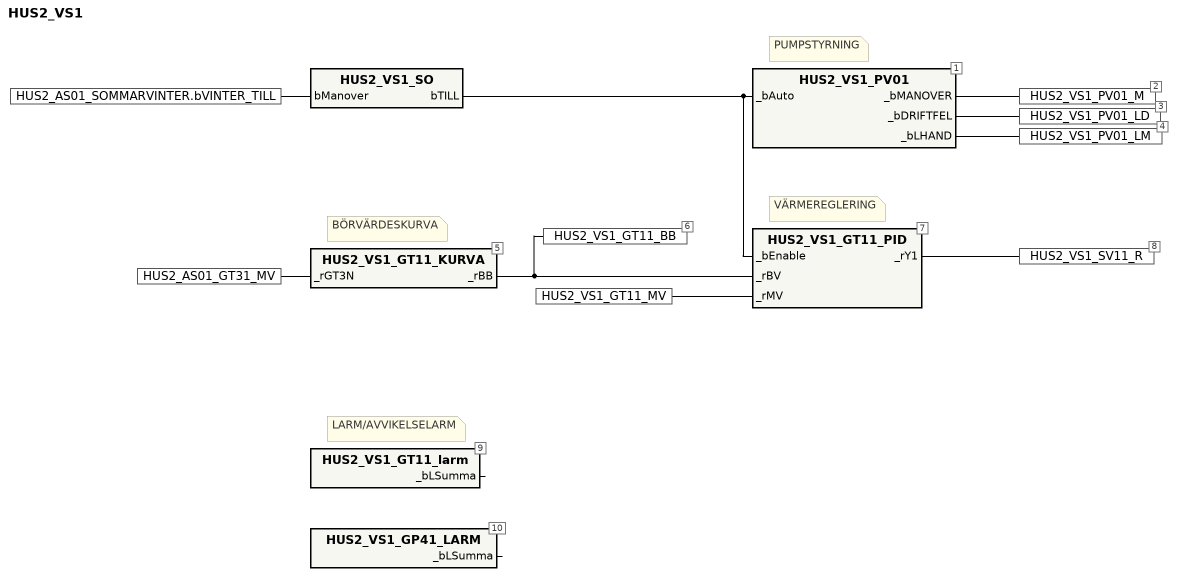
_CFC_ (* Continuous Function Chart, elements in execution order *)
(* LARM/AVVIKELSELARM *)
(* BÖRVÄRDESKURVA *)
(* PUMPSTYRNING *)
(* VÄRMEREGLERING *)
#0 HUS2_VS1_SO(bManover: HUS2_AS01_SOMMARVINTER.bVINTER_TILL)
#1 HUS2_VS1_PV01(_bAuto: #0.bTILL)
#2 HUS2_VS1_PV01_M <= #1._bMANOVER
#3 HUS2_VS1_PV01_LD <= #1._bDRIFTFEL
#4 HUS2_VS1_PV01_LM <= #1._bLHAND
#5 HUS2_VS1_GT11_KURVA(_rGT3N: HUS2_AS01_GT31_MV)
#6 HUS2_VS1_GT11_BB <= #5._rBB
#7 HUS2_VS1_GT11_PID(_bEnable: #0.bTILL, _rBV: #5._rBB, _rMV: HUS2_VS1_GT11_MV)
#8 HUS2_VS1_SV11_R <= #7._rY1
#9 HUS2_VS1_GT11_larm()
#10 HUS2_VS1_GP41_LARM()
_END_CFC_
(* the same logic as Structured Text *)
(* LARM/AVVIKELSELARM *)
(* BÖRVÄRDESKURVA *)
(* PUMPSTYRNING *)
(* VÄRMEREGLERING *)
HUS2_VS1_SO(bManover := HUS2_AS01_SOMMARVINTER.bVINTER_TILL);
HUS2_VS1_PV01(_bAuto := HUS2_VS1_SO.bTILL);
HUS2_VS1_PV01_M := HUS2_VS1_PV01._bMANOVER;
HUS2_VS1_PV01_LD := HUS2_VS1_PV01._bDRIFTFEL;
HUS2_VS1_PV01_LM := HUS2_VS1_PV01._bLHAND;
HUS2_VS1_GT11_KURVA(_rGT3N := HUS2_AS01_GT31_MV);
HUS2_VS1_GT11_BB := HUS2_VS1_GT11_KURVA._rBB;
HUS2_VS1_GT11_PID(_bEnable := HUS2_VS1_SO.bTILL, _rBV := HUS2_VS1_GT11_KURVA._rBB, _rMV := HUS2_VS1_GT11_MV);
HUS2_VS1_SV11_R := HUS2_VS1_GT11_PID._rY1;
HUS2_VS1_GT11_larm();
HUS2_VS1_GP41_LARM();
END_PROGRAM

(* POU SYSTEM/VS1/HUS2_VS1_SO, CFC *)
PROGRAM HUS2_VS1_SO
VAR_INPUT

	bManover: BOOL;
END_VAR

VAR
	SERVICEOMKOPPLARE: fbManualOverride;

	UPPSTARTSSEKVENSIERING: BOOL:=TRUE;
END_VAR

VAR_OUTPUT
	bTILL:BOOL;

END_VAR
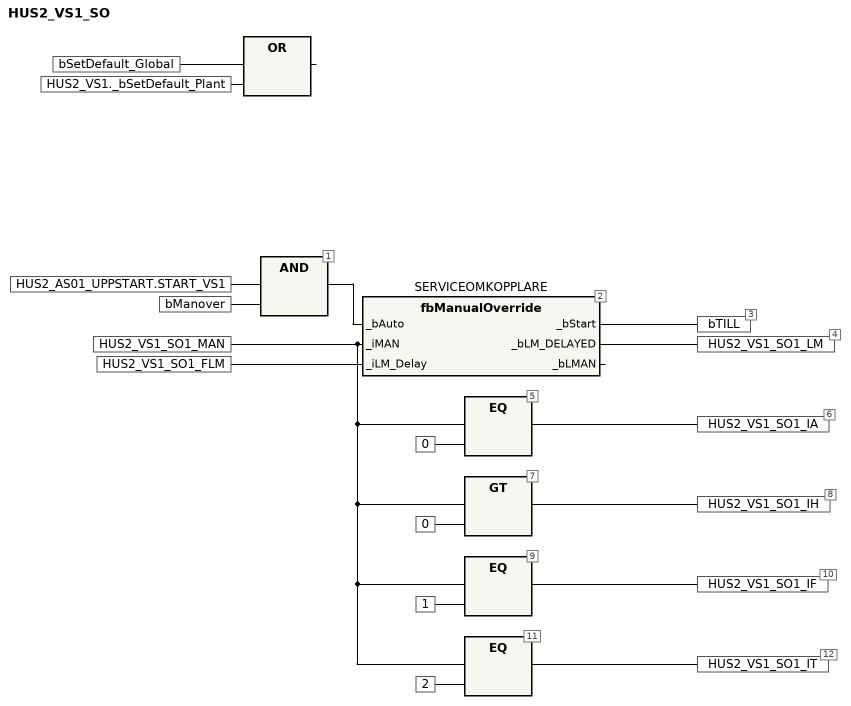
_CFC_ (* Continuous Function Chart, elements in execution order *)
#0 OR(bSetDefault_Global, HUS2_VS1._bSetDefault_Plant)
#1 AND(HUS2_AS01_UPPSTART.START_VS1, bManover)
#2 SERVICEOMKOPPLARE:fbManualOverride(_bAuto: #1, _iMAN: HUS2_VS1_SO1_MAN, _iLM_Delay: HUS2_VS1_SO1_FLM)
#3 bTILL <= #2._bStart
#4 HUS2_VS1_SO1_LM <= #2._bLM_DELAYED
#5 EQ(HUS2_VS1_SO1_MAN, 0)
#6 HUS2_VS1_SO1_IA <= #5
#7 GT(HUS2_VS1_SO1_MAN, 0)
#8 HUS2_VS1_SO1_IH <= #7
#9 EQ(HUS2_VS1_SO1_MAN, 1)
#10 HUS2_VS1_SO1_IF <= #9
#11 EQ(HUS2_VS1_SO1_MAN, 2)
#12 HUS2_VS1_SO1_IT <= #11
_END_CFC_
(* the same logic as Structured Text *)
(* result unused: bSetDefault_Global OR HUS2_VS1._bSetDefault_Plant *)
SERVICEOMKOPPLARE(_bAuto := HUS2_AS01_UPPSTART.START_VS1 AND bManover, _iMAN := HUS2_VS1_SO1_MAN, _iLM_Delay := HUS2_VS1_SO1_FLM);
bTILL := SERVICEOMKOPPLARE._bStart;
HUS2_VS1_SO1_LM := SERVICEOMKOPPLARE._bLM_DELAYED;
HUS2_VS1_SO1_IA := HUS2_VS1_SO1_MAN = 0;
HUS2_VS1_SO1_IH := HUS2_VS1_SO1_MAN > 0;
HUS2_VS1_SO1_IF := HUS2_VS1_SO1_MAN = 1;
HUS2_VS1_SO1_IT := HUS2_VS1_SO1_MAN = 2;
END_PROGRAM

(* POU SYSTEM/VS1/Pumpstyrning/HUS2_VS1_PV01, CFC *)
PROGRAM HUS2_VS1_PV01

VAR

	Default: BOOL;
	Motor: FB_HVACMotor1Speed;

	fbReset1: fbBool_Reset;
	AlarmDelay: fbDelayedAlarmSeconds;

	MANHAND: fbManualOverride;
END_VAR
VAR


(********************MOTOR********************)
(*INPUT*)
	eCtrlModeActuator			:E_HVACActuatorMode;
	tStartDelay						:TIME;
	tStopDelay						:TIME;
	tDelayFeedbContactor			:TIME:=T#30s;
	tFeedbProcessTimer				:TIME:=T#30s;
	tDelayFeedbProcess				:TIME:=T#30s;
(*OUTPUT*)
	byState							:BYTE ;
	bStateAuto							:BOOL;
	bStateRepairSwitch				:BOOL;
	bStateManSwitch				:BOOL;
	eStateModeActuator				:E_HVACActuatorMode;
	byError							:BYTE ;
	bErrorMotorprotec				:BOOL;
	bErrorFeedbContactor			:BOOL;
	bErrorFeedbProcess			:BOOL;
	bInvalidParameter				:BOOL;


END_VAR

VAR_INPUT
	_bAuto							:BOOL;(* enable function block *)
END_VAR

VAR_OUTPUT
	_bMANOVER						:BOOL;
	_bDRIFTFEL						:BOOL;
	_bLHAND							:BOOL;
END_VAR
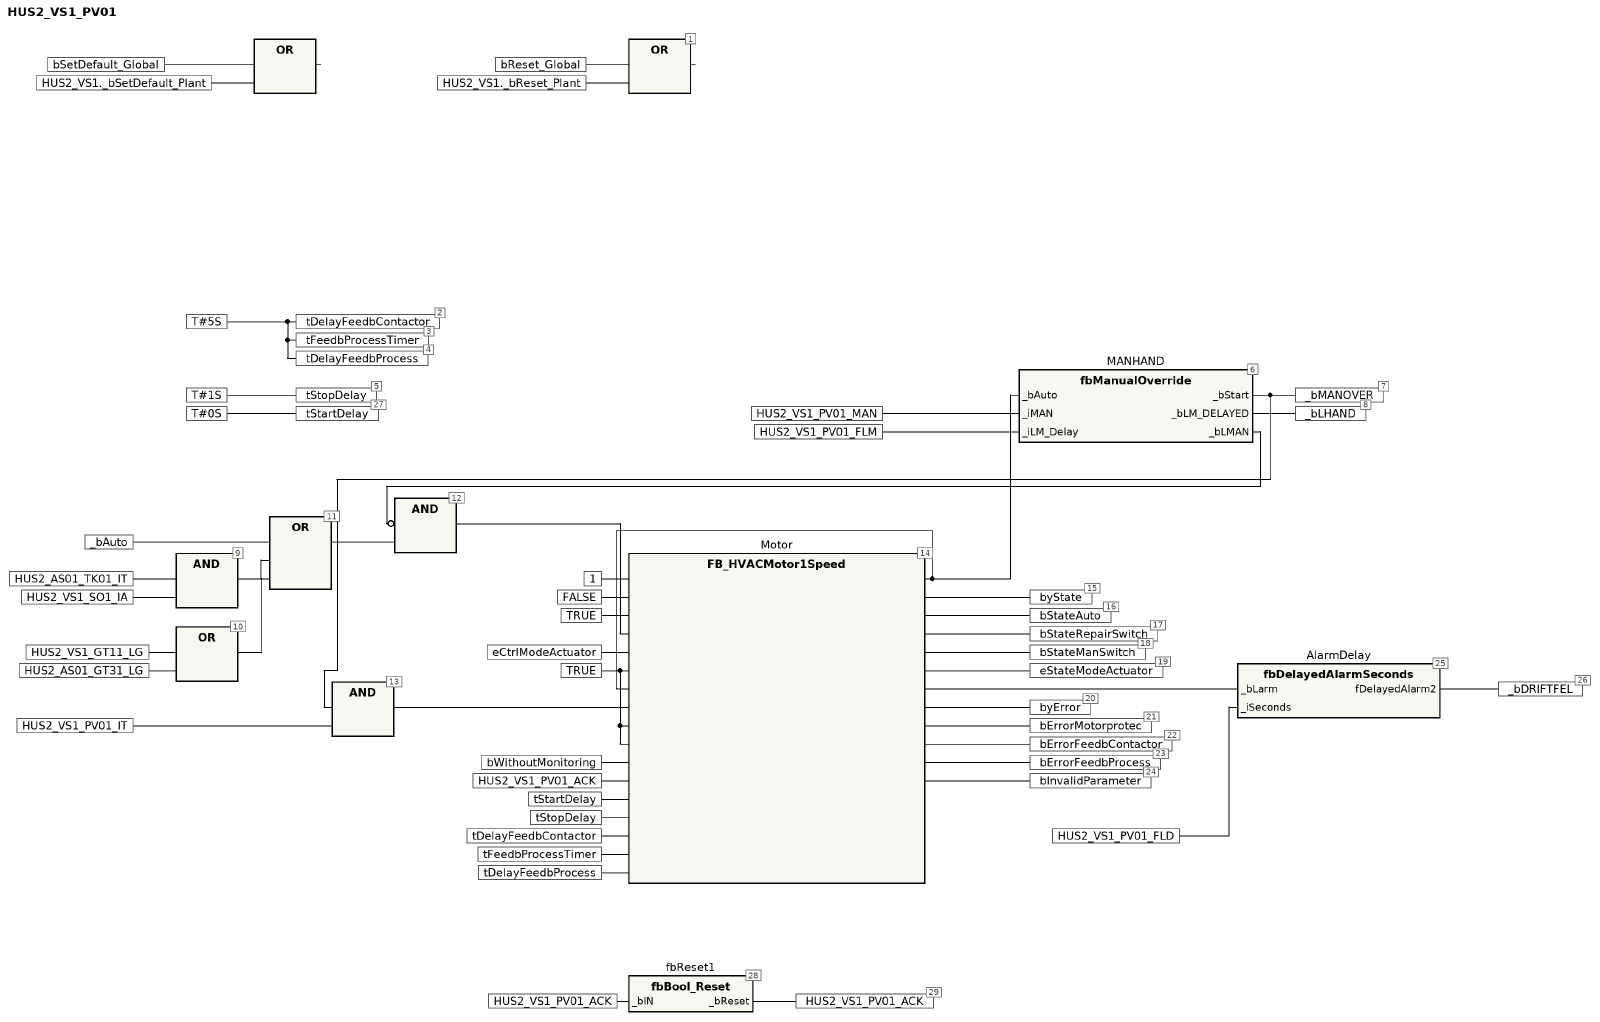
_CFC_ (* Continuous Function Chart, elements in execution order *)
#0 OR(bSetDefault_Global, HUS2_VS1._bSetDefault_Plant)
#1 OR(bReset_Global, HUS2_VS1._bReset_Plant)
#2 tDelayFeedbContactor <= T#5S
#3 tFeedbProcessTimer <= T#5S
#4 tDelayFeedbProcess <= T#5S
#5 tStopDelay <= T#1S
#6 MANHAND:fbManualOverride(_bAuto: #14.out 1, _iMAN: HUS2_VS1_PV01_MAN, _iLM_Delay: HUS2_VS1_PV01_FLM)
#7 _bMANOVER <= #6._bStart
#8 _bLHAND <= #6._bLM_DELAYED
#9 AND(HUS2_AS01_TK01_IT, HUS2_VS1_SO1_IA)
#10 OR(HUS2_VS1_GT11_LG, HUS2_AS01_GT31_LG)
#11 OR(_bAuto, #9, #10)
#12 AND(NOT #6._bLMAN, #11)
#13 AND(#6._bStart, HUS2_VS1_PV01_IT)
#14 Motor:FB_HVACMotor1Speed(1, FALSE, TRUE, #12, eCtrlModeActuator, TRUE, #14.out 1, #13, TRUE, TRUE, bWithoutMonitoring, HUS2_VS1_PV01_ACK, tStartDelay, tStopDelay, tDelayFeedbContactor, tFeedbProcessTimer, tDelayFeedbProcess)
#15 byState <= #14.out 2
#16 bStateAuto <= #14.out 3
#17 bStateRepairSwitch <= #14.out 4
#18 bStateManSwitch <= #14.out 5
#19 eStateModeActuator <= #14.out 6
#20 byError <= #14.out 8
#21 bErrorMotorprotec <= #14.out 9
#22 bErrorFeedbContactor <= #14.out 10
#23 bErrorFeedbProcess <= #14.out 11
#24 bInvalidParameter <= #14.out 12
#25 AlarmDelay:fbDelayedAlarmSeconds(_bLarm: #14.out 7, _iSeconds: HUS2_VS1_PV01_FLD)
#26 _bDRIFTFEL <= #25.fDelayedAlarm2
#27 tStartDelay <= T#0S
#28 fbReset1:fbBool_Reset(_bIN: HUS2_VS1_PV01_ACK)
#29 HUS2_VS1_PV01_ACK <= #28._bReset
_END_CFC_
END_PROGRAM

(* POU SYSTEM/VS1/Börvärden & kurvor/HUS2_VS1_GT11_KURVA, FAI *)
PROGRAM HUS2_VS1_GT11_KURVA
VAR
(****************************************** heating curve **********************************************************************************************************************)

	_bSetDefaultHC			:BOOL;


	fbScale_n:			FB_HVACScale_nPoint;
	_bErrParam:			BOOL;								(*ParameterError*)
	stScaleParameter:	ST_HVACParameterScale_nPoint	;	(*Parameter struktur på antal brutpunkter*)


	fbTemp1:	FB_HVACPersistent_Real;
	fbTemp2:	FB_HVACPersistent_Real;
	fbTemp3:	FB_HVACPersistent_Real;
	fbTemp4:	FB_HVACPersistent_Real;
	fbTemp5:	FB_HVACPersistent_Real;

	fbOutsideTemp1:	FB_HVACPersistent_Real;
	fbOutsideTemp2:	FB_HVACPersistent_Real;
	fbOutsideTemp3:	FB_HVACPersistent_Real;
	fbOutsideTemp4:	FB_HVACPersistent_Real;
	fbOutsideTemp5:	FB_HVACPersistent_Real;
	BB_min: FB_HVACPersistent_Real;
	BB_max: FB_HVACPersistent_Real;

END_VAR

VAR_INPUT
	_rGT3N	:REAL; (*Utegivare*)

END_VAR

VAR_OUTPUT
	_rBB		:LREAL;
END_VAR
(* body not read: cfc97 *)
END_PROGRAM

(* POU SYSTEM/VS1/Tempreglering/HUS2_VS1_GT11_PID, FAI *)
PROGRAM HUS2_VS1_GT11_PID

VAR_INPUT
	_bEnable		:BOOL;
	_rBV			:REAL;
	_rMV			:REAL;

END_VAR

VAR_OUTPUT
	_rY1                         : REAL;
END_VAR


VAR
	_bSetDefaultPID:BOOL;
	_bReset_Local:BOOL;


	SVX: FB_HVACPIDCtrl;
	eDataSecurityType         : E_HVACDataSecurityType;
	rInitialValue            : REAL;
	bResetController          : BOOL;
	_eCtrlMode				:E_HVACCtrlMode;(*
									eHVACCtrlMode_Auto      := 0,
								   	eHVACCtrlMode_Manual   := 1 *)
	_rOverrideValue			:REAL;(* controller output rY in operating mode eCtrlMode =1 *)
	rXW                        : REAL;
	bMaxLimit                  : BOOL;
	bMinLimit                  : BOOL;
	bActive                    : BOOL;
	bARWactive                 : BOOL;
	eState                     : E_HVACState;
	bError                     : BOOL;
	eErrorCode                 : E_HVACErrorCodes;
	bInvalidParameter          : BOOL;

	bDirection              : BOOL;
	_rKP: REAL;
	_rCH: REAL;
	tTi                     : TIME;
	tTv                     : TIME;
	tTd                     : TIME;

	rYMin                   : REAL;
	rYMax                   : REAL;

	CI: fbBer_PID_inst;
	CS: fbBer_PID_inst;
	CD: fbBer_PID_inst;

	fbPersistent_CH: FB_HVACPersistent_Real;
	fbPersistent_CP: FB_HVACPersistent_Real;
	fbPersistent_CI: FB_HVACPersistent_Real;
	fbPersistent_CS: FB_HVACPersistent_Real;
	fbPersistent_CD: FB_HVACPersistent_Real;
	LM_DELAY: fbDelayedAlarmMinutes;
END_VAR
(* body not read: cfc97 *)
END_PROGRAM

(* POU SYSTEM/VS1/Larm/HUS2_VS1_GT11_LARM, FAI *)
PROGRAM HUS2_VS1_GT11_LARM

VAR_OUTPUT
	_bLSumma					: BOOL;	(*Summalarm*)

END_VAR
VAR

	_bSetDefault: 				BOOL;		(*Se default values*)
	fbLarm: fbAvvikelselarm;


	fbHigh: FB_HVACPersistent_Real;
	fbAlarmDelayLH: FB_HVACPersistent_Int;
	fbLow: FB_HVACPersistent_Real;
	fbAlarmDelayLL: FB_HVACPersistent_Int;


END_VAR
(* body not read: cfc97 *)
END_PROGRAM

(* POU xEgna Funktionsblock/fbAvvikelselarm, CFC *)
FUNCTION_BLOCK fbAvvikelselarm
VAR
	TON1: TON;
	TON2: TON;
END_VAR
VAR_INPUT
	_rBB: REAL;
	_rMV: REAL;
	_rLL: REAL;
	_iFLL: INT;
	_rLH: REAL;
	_iFLH: INT;
	_bAktiveraLarm: BOOL;

END_VAR


VAR_OUTPUT
	_bLL: BOOL;
	_bLH: BOOL;
	_bLSummA: BOOL;
END_VAR
VAR (* helpers for the ST form of the networks *)
	_t54 : TIME;
END_VAR
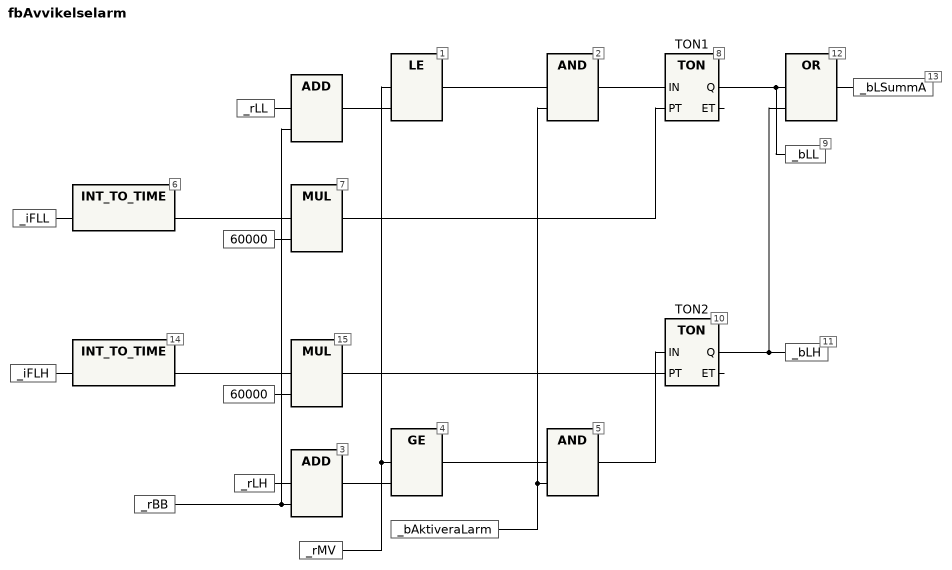
_CFC_ (* Continuous Function Chart, elements in execution order *)
#0 ADD(_rLL, _rBB)
#1 LE(_rMV, #0)
#2 AND(#1, _bAktiveraLarm)
#3 ADD(_rLH, _rBB)
#4 GE(_rMV, #3)
#5 AND(#4, _bAktiveraLarm)
#6 INT_TO_TIME(_iFLL)
#7 MUL(#6, 60000)
#8 TON1:TON(IN: #2, PT: #7)
#9 _bLL <= #8.Q
#10 TON2:TON(IN: #5, PT: #15)
#11 _bLH <= #10.Q
#12 OR(#8.Q, #10.Q)
#13 _bLSummA <= #12
#14 INT_TO_TIME(_iFLH)
#15 MUL(#14, 60000)
_END_CFC_
(* the same logic as Structured Text *)
TON1(IN := (_rMV <= (_rLL + _rBB)) AND _bAktiveraLarm, PT := INT_TO_TIME(_iFLL) * 60000);
_bLL := TON1.Q;
TON2(IN := (_rMV >= (_rLH + _rBB)) AND _bAktiveraLarm, PT := _t54);
_bLH := TON2.Q;
_bLSummA := TON1.Q OR TON2.Q;
_t54 := INT_TO_TIME(_iFLH) * 60000;
END_FUNCTION_BLOCK

(* POU SYSTEM/VS1/Larm/HUS2_VS1_GP41_LARM, FAI *)
PROGRAM HUS2_VS1_GP41_LARM

VAR_OUTPUT
	_bLSumma					: BOOL;	(*Summalarm*)

END_VAR
VAR

	_bSetDefault: 				BOOL;		(*Se default values*)
	fbLarm: fbAvvikelselarm;
	fbLow: FB_HVACPersistent_Real;
	fbAlarmDelayLL: FB_HVACPersistent_Int;
	fbHigh: FB_HVACPersistent_Real;
	fbAlarmDelayLH: FB_HVACPersistent_Int;
END_VAR
(* body not read: cfc97 *)
END_PROGRAM

(* POU SYSTEM/VV1/HUS2_VV1, CFC *)
PROGRAM HUS2_VV1
VAR
	_bSetDefault_Plant		:BOOL;
	_bReset_Plant				:BOOL;

	VV_BV: FB_HVACPersistent_Real;
END_VAR
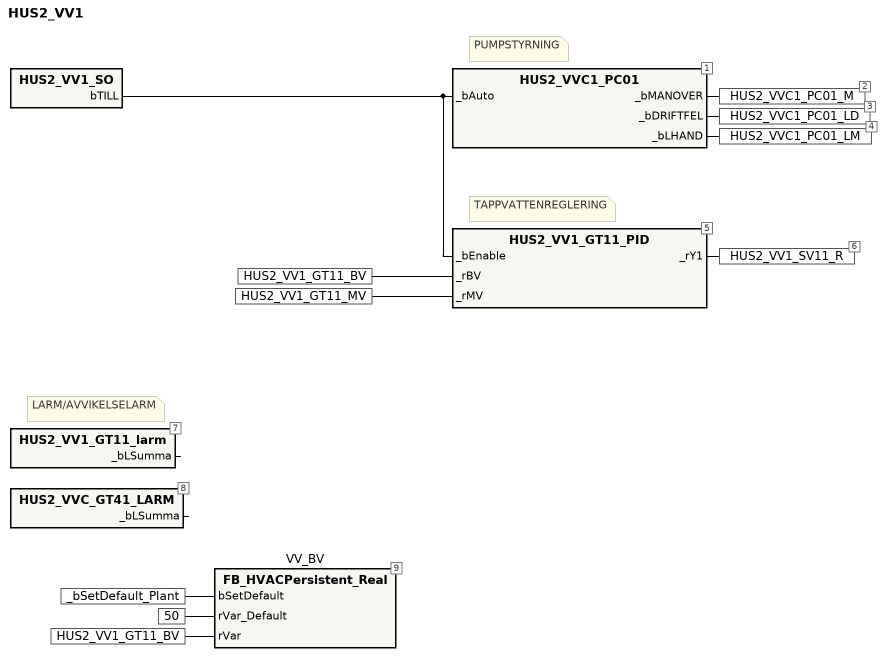
_CFC_ (* Continuous Function Chart, elements in execution order *)
(* TAPPVATTENREGLERING *)
(* PUMPSTYRNING *)
(* LARM/AVVIKELSELARM *)
#0 HUS2_VV1_SO()
#1 HUS2_VVC1_PC01(_bAuto: #0.bTILL)
#2 HUS2_VVC1_PC01_M <= #1._bMANOVER
#3 HUS2_VVC1_PC01_LD <= #1._bDRIFTFEL
#4 HUS2_VVC1_PC01_LM <= #1._bLHAND
#5 HUS2_VV1_GT11_PID(_bEnable: #0.bTILL, _rBV: HUS2_VV1_GT11_BV, _rMV: HUS2_VV1_GT11_MV)
#6 HUS2_VV1_SV11_R <= #5._rY1
#7 HUS2_VV1_GT11_larm()
#8 HUS2_VVC_GT41_LARM()
#9 VV_BV:FB_HVACPersistent_Real(bSetDefault: _bSetDefault_Plant, rVar_Default: 50, rVar: HUS2_VV1_GT11_BV)
_END_CFC_
(* the same logic as Structured Text *)
(* TAPPVATTENREGLERING *)
(* PUMPSTYRNING *)
(* LARM/AVVIKELSELARM *)
HUS2_VV1_SO();
HUS2_VVC1_PC01(_bAuto := HUS2_VV1_SO.bTILL);
HUS2_VVC1_PC01_M := HUS2_VVC1_PC01._bMANOVER;
HUS2_VVC1_PC01_LD := HUS2_VVC1_PC01._bDRIFTFEL;
HUS2_VVC1_PC01_LM := HUS2_VVC1_PC01._bLHAND;
HUS2_VV1_GT11_PID(_bEnable := HUS2_VV1_SO.bTILL, _rBV := HUS2_VV1_GT11_BV, _rMV := HUS2_VV1_GT11_MV);
HUS2_VV1_SV11_R := HUS2_VV1_GT11_PID._rY1;
HUS2_VV1_GT11_larm();
HUS2_VVC_GT41_LARM();
VV_BV(bSetDefault := _bSetDefault_Plant, rVar_Default := 50, rVar := HUS2_VV1_GT11_BV);
END_PROGRAM

(* POU SYSTEM/VV1/HUS2_VV1_SO, CFC *)
PROGRAM HUS2_VV1_SO

VAR

	LM_DELAY: fbDelayedAlarmMinutes;
END_VAR

VAR_OUTPUT
	bTILL:BOOL;

END_VAR
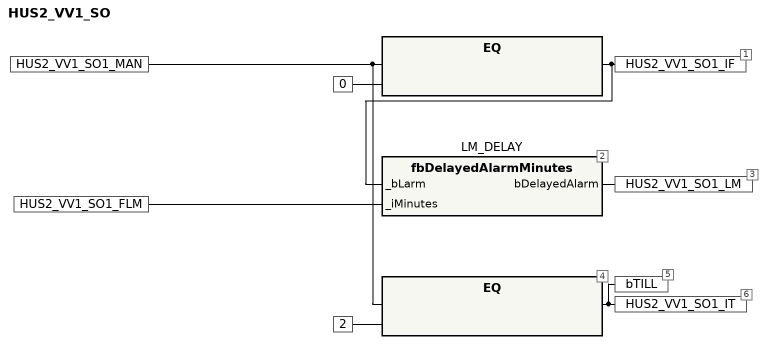
_CFC_ (* Continuous Function Chart, elements in execution order *)
#0 EQ(HUS2_VV1_SO1_MAN, 0)
#1 HUS2_VV1_SO1_IF <= #0
#2 LM_DELAY:fbDelayedAlarmMinutes(_bLarm: #0, _iMinutes: HUS2_VV1_SO1_FLM)
#3 HUS2_VV1_SO1_LM <= #2.bDelayedAlarm
#4 EQ(HUS2_VV1_SO1_MAN, 2)
#5 bTILL <= #4
#6 HUS2_VV1_SO1_IT <= #4
_END_CFC_
(* the same logic as Structured Text *)
HUS2_VV1_SO1_IF := HUS2_VV1_SO1_MAN = 0;
LM_DELAY(_bLarm := HUS2_VV1_SO1_MAN = 0, _iMinutes := HUS2_VV1_SO1_FLM);
HUS2_VV1_SO1_LM := LM_DELAY.bDelayedAlarm;
bTILL := HUS2_VV1_SO1_MAN = 2;
HUS2_VV1_SO1_IT := HUS2_VV1_SO1_MAN = 2;
END_PROGRAM

(* POU SYSTEM/VV1/Pumpstyrning/HUS2_VVC1_PC01, CFC *)
PROGRAM HUS2_VVC1_PC01

VAR

	Default: BOOL;
	Motor: FB_HVACMotor1Speed;

	fbReset1: fbBool_Reset;
	AlarmDelay: fbDelayedAlarmSeconds;

	MANHAND: fbManualOverride;
END_VAR
VAR


(********************MOTOR********************)
(*INPUT*)
	eCtrlModeActuator			:E_HVACActuatorMode;
	tStartDelay						:TIME;
	tStopDelay						:TIME;
	tDelayFeedbContactor			:TIME:=T#30s;
	tFeedbProcessTimer				:TIME:=T#30s;
	tDelayFeedbProcess				:TIME:=T#30s;
(*OUTPUT*)
	byState							:BYTE ;
	bStateAuto							:BOOL;
	bStateRepairSwitch				:BOOL;
	bStateManSwitch				:BOOL;
	eStateModeActuator				:E_HVACActuatorMode;
	byError							:BYTE ;
	bErrorMotorprotec				:BOOL;
	bErrorFeedbContactor			:BOOL;
	bErrorFeedbProcess			:BOOL;
	bInvalidParameter				:BOOL;


END_VAR

VAR_INPUT
	_bAuto							:BOOL;(* enable function block *)
END_VAR

VAR_OUTPUT
	_bMANOVER						:BOOL;
	_bDRIFTFEL						:BOOL;
	_bLHAND							:BOOL;
END_VAR
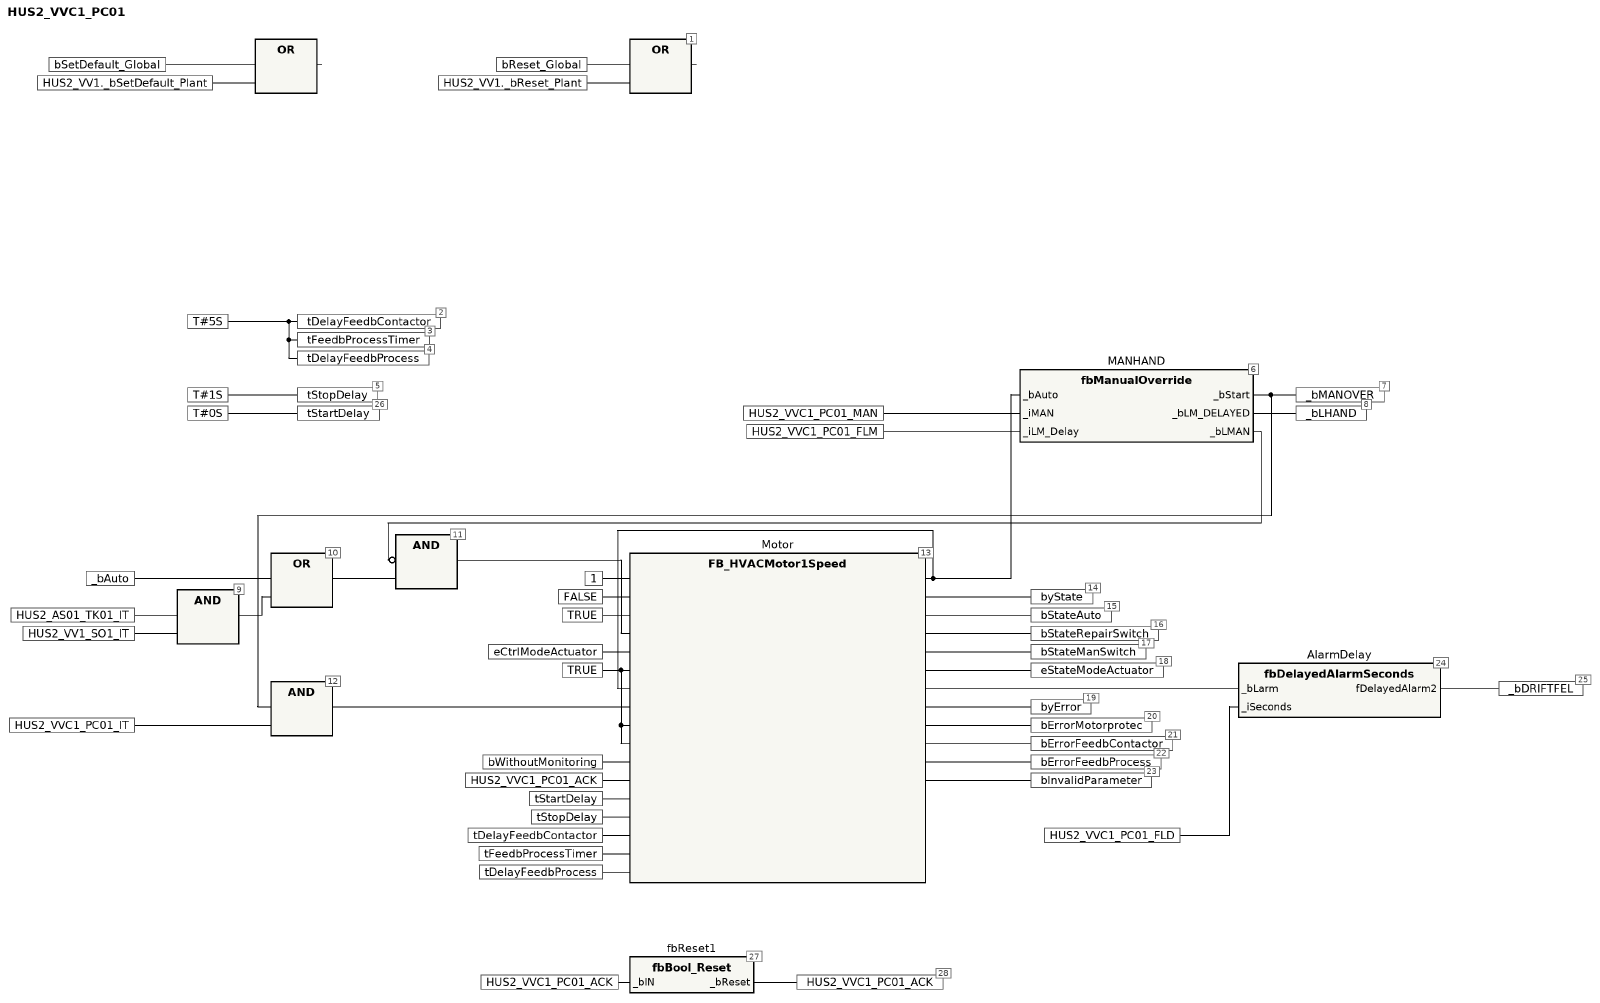
_CFC_ (* Continuous Function Chart, elements in execution order *)
#0 OR(bSetDefault_Global, HUS2_VV1._bSetDefault_Plant)
#1 OR(bReset_Global, HUS2_VV1._bReset_Plant)
#2 tDelayFeedbContactor <= T#5S
#3 tFeedbProcessTimer <= T#5S
#4 tDelayFeedbProcess <= T#5S
#5 tStopDelay <= T#1S
#6 MANHAND:fbManualOverride(_bAuto: #13.out 1, _iMAN: HUS2_VVC1_PC01_MAN, _iLM_Delay: HUS2_VVC1_PC01_FLM)
#7 _bMANOVER <= #6._bStart
#8 _bLHAND <= #6._bLM_DELAYED
#9 AND(HUS2_AS01_TK01_IT, HUS2_VV1_SO1_IT)
#10 OR(_bAuto, #9)
#11 AND(NOT #6._bLMAN, #10)
#12 AND(#6._bStart, HUS2_VVC1_PC01_IT)
#13 Motor:FB_HVACMotor1Speed(1, FALSE, TRUE, #11, eCtrlModeActuator, TRUE, #13.out 1, #12, TRUE, TRUE, bWithoutMonitoring, HUS2_VVC1_PC01_ACK, tStartDelay, tStopDelay, tDelayFeedbContactor, tFeedbProcessTimer, tDelayFeedbProcess)
#14 byState <= #13.out 2
#15 bStateAuto <= #13.out 3
#16 bStateRepairSwitch <= #13.out 4
#17 bStateManSwitch <= #13.out 5
#18 eStateModeActuator <= #13.out 6
#19 byError <= #13.out 8
#20 bErrorMotorprotec <= #13.out 9
#21 bErrorFeedbContactor <= #13.out 10
#22 bErrorFeedbProcess <= #13.out 11
#23 bInvalidParameter <= #13.out 12
#24 AlarmDelay:fbDelayedAlarmSeconds(_bLarm: #13.out 7, _iSeconds: HUS2_VVC1_PC01_FLD)
#25 _bDRIFTFEL <= #24.fDelayedAlarm2
#26 tStartDelay <= T#0S
#27 fbReset1:fbBool_Reset(_bIN: HUS2_VVC1_PC01_ACK)
#28 HUS2_VVC1_PC01_ACK <= #27._bReset
_END_CFC_
END_PROGRAM

(* POU SYSTEM/VV1/Tempreglering/HUS2_VV1_GT11_PID, FAI *)
PROGRAM HUS2_VV1_GT11_PID

VAR_INPUT
	_bEnable		:BOOL;
	_rBV			:REAL;
	_rMV			:REAL;
END_VAR

VAR_OUTPUT
	_rY1                         : REAL;
END_VAR


VAR
	_bSetDefaultPID:BOOL;
	_bReset_Local:BOOL;


	SVX: FB_HVACPIDCtrl;
	eDataSecurityType         : E_HVACDataSecurityType;
	rInitialValue            : REAL;
	bResetController          : BOOL;
	_eCtrlMode				:E_HVACCtrlMode;(*
									eHVACCtrlMode_Auto      := 0,
								   	eHVACCtrlMode_Manual   := 1 *)
	_rOverrideValue			:REAL;(* controller output rY in operating mode eCtrlMode =1 *)
	rXW                        : REAL;
	bMaxLimit                  : BOOL;
	bMinLimit                  : BOOL;
	bActive                    : BOOL;
	bARWactive                 : BOOL;
	eState                     : E_HVACState;
	bError                     : BOOL;
	eErrorCode                 : E_HVACErrorCodes;
	bInvalidParameter          : BOOL;

	bDirection              : BOOL;
	_rKP: REAL;
	_rCH: REAL;
	tTi                     : TIME;
	tTv                     : TIME;
	tTd                     : TIME;

	rYMin                   : REAL;
	rYMax                   : REAL;

	CI: fbBer_PID_inst;
	CS: fbBer_PID_inst;
	CD: fbBer_PID_inst;

	fbPersistent_CH: FB_HVACPersistent_Real;
	fbPersistent_CP: FB_HVACPersistent_Real;
	fbPersistent_CI: FB_HVACPersistent_Real;
	fbPersistent_CS: FB_HVACPersistent_Real;
	fbPersistent_CD: FB_HVACPersistent_Real;
	LM_DELAY: fbDelayedAlarmMinutes;
END_VAR
(* body not read: cfc97 *)
END_PROGRAM

(* POU SYSTEM/VV1/Larm/HUS2_VV1_GT11_LARM, FAI *)
PROGRAM HUS2_VV1_GT11_LARM

VAR_OUTPUT
	_bLSumma					: BOOL;	(*Summalarm*)

END_VAR
VAR

	_bSetDefault: 				BOOL;		(*Se default values*)
	fbLarm: fbAvvikelselarm;


	fbHigh: FB_HVACPersistent_Real;
	fbAlarmDelayLH: FB_HVACPersistent_Int;
	fbLow: FB_HVACPersistent_Real;
	fbAlarmDelayLL: FB_HVACPersistent_Int;


END_VAR
(* body not read: cfc97 *)
END_PROGRAM

(* POU SYSTEM/VV1/Larm/HUS2_VVC_GT41_LARM, FAI *)
PROGRAM HUS2_VVC_GT41_LARM

VAR_OUTPUT
	_bLSumma					: BOOL;	(*Summalarm*)

END_VAR
VAR

	_bSetDefault: 				BOOL;		(*Se default values*)
	fbLarm: fbAvvikelselarm;


	fbHigh: FB_HVACPersistent_Real;
	fbAlarmDelayLH: FB_HVACPersistent_Int;


END_VAR
(* body not read: cfc97 *)
END_PROGRAM

(* POU SYSTEM/VS20/HUS1_VS20, CFC *)
PROGRAM HUS1_VS20
VAR
	_bSetDefault_Plant		:BOOL;
	_bReset_Plant				:BOOL;

END_VAR
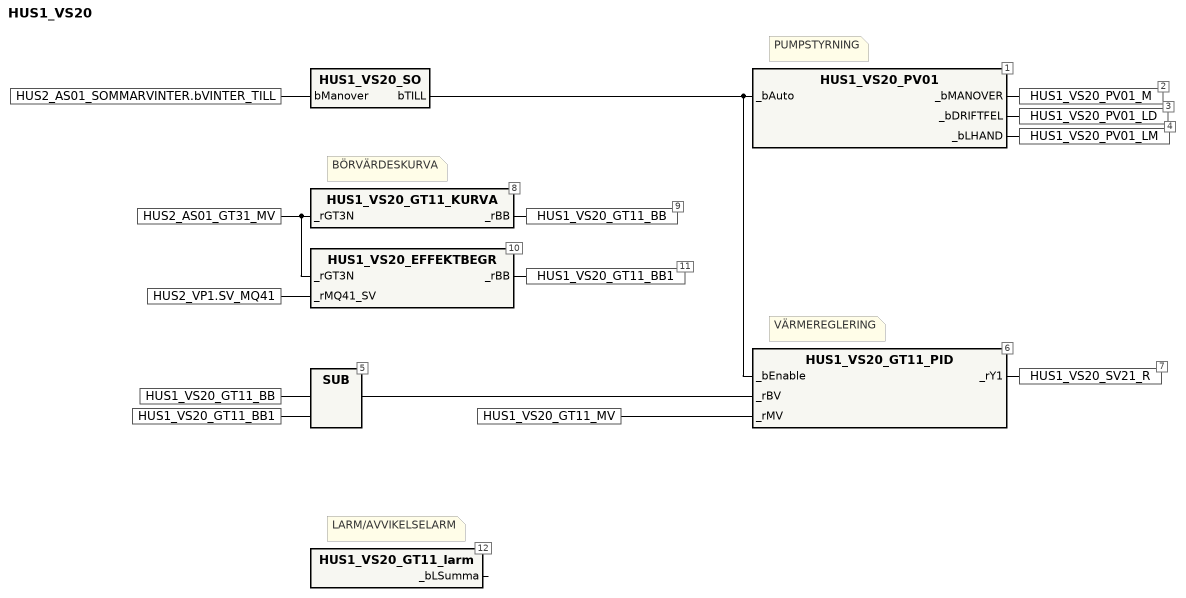
